    (*Switch to another storage tank with same varnish if storage tank reaches error level.*)
    IF iL_StoragetankAssignmentIndex[iL_Counter] <> 0 THEN
      IF sAdsIkInkStorageTank[iL_StoragetankAssignmentIndex[iL_Counter]].bO_StorageTankError THEN
        FOR iL_Counter2 := 1 TO iCIk_NB_INKSTORAGE_TANK DO
          IF     (iL_StoragetankAssignmentIndex[iL_Counter] <> iL_Counter2)
             AND (  sAdsIkInkStorageTank[iL_StoragetankAssignmentIndex[iL_Counter]].sI_InkParameter.iIndex
                  = sAdsIkInkStorageTank[iL_Counter2].sI_InkParameter.iIndex)
             AND NOT sAdsIkInkStorageTank[iL_Counter2].bO_StorageTankError
          THEN
            sAdsIkHeaderTank[iL_Counter].sI_StoragetankAssignment   .lI_Val := UDINT_TO_DINT(sL_BLK_INKSTORAGE_TANK[iL_Counter2].iBlk_AdsId);
            sAdsIkHeaderTank[iL_Counter].sO_ActStoragetankAssignment.lI_Val := UDINT_TO_DINT(sL_BLK_INKSTORAGE_TANK[iL_Counter2].iBlk_AdsId);
          END_IF
        END_FOR
      END_IF
    END_IF
  
    (*Check assignment of header tank to storage tank*)
    iL_StoragetankAssignmentIndex   [iL_Counter] := 0;
    iL_ActStoragetankAssignmentIndex[iL_Counter] := 0;
  
    FOR iL_Counter2 := 1 TO iCIk_NB_INKSTORAGE_TANK DO
      IF   sAdsIkHeaderTank[iL_Counter].sI_StoragetankAssignment.lI_Val
         = UDINT_TO_DINT(sL_BLK_INKSTORAGE_TANK[iL_Counter2].iBlk_AdsId)
      THEN
        iL_StoragetankAssignmentIndex[iL_Counter] := iL_Counter2;
      END_IF
  
      IF   sAdsIkHeaderTank[iL_Counter].sO_ActStoragetankAssignment.lI_Val
         = UDINT_TO_DINT(sL_BLK_INKSTORAGE_TANK[iL_Counter2].iBlk_AdsId)
      THEN
        iL_ActStoragetankAssignmentIndex[iL_Counter] := iL_Counter2;
      END_IF
    END_FOR

    (*Purge: outflow valve while DeAir*)
    bL_PurgeOutflow2ValveHT[iL_Counter] :=     fb_PurgeController[iCIk_MAP_HEADERTANK_PURGE_CONTR[iL_Counter]].fb_PurgeContr.bI_DeAirSelect[iCIk_MAP_HEADERTANK_PURGE_GROUPIDX[iL_Counter]]
                                           AND fb_PurgeController[iCIk_MAP_HEADERTANK_PURGE_CONTR[iL_Counter]].fb_PurgeContr.bO_Outflow2Valve;

  END_FOR
  
  
  
  FOR iL_Counter := 1 TO iCIk_NB_HEADERTANK DO
    (*Data from assigned storage tank*)
    IF     (iL_ActStoragetankAssignmentIndex[iL_Counter] > 0)
       AND (iL_ActStoragetankAssignmentIndex[iL_Counter] <= iCIk_NB_INKSTORAGE_TANK)
    THEN
      fL_StorageTankLevelLiter := sAdsIkInkStorageTank[iL_ActStoragetankAssignmentIndex[iL_Counter]].fO_StorageTankLevelLiter.fO_Val;
  
      IF sAdsIkInkStorageTank[iL_ActStoragetankAssignmentIndex[iL_Counter]].sI_InkParameter.iTimer = 0 THEN
        IF (sAdsIkInkStorageTank[iL_ActStoragetankAssignmentIndex[iL_Counter]].sI_InkParameter.iColorId >= 254) THEN
          tL_TimeReturnFlow := tL_TimeReturnFlowHt[iL_Counter];
        ELSE
          tL_TimeReturnFlow := UDINT_TO_TIME(lL_TimeReturnFlow * 1000);
        END_IF
      ELSE
        tL_TimeReturnFlow := UDINT_TO_TIME(UINT_TO_UDINT(sAdsIkInkStorageTank[iL_ActStoragetankAssignmentIndex[iL_Counter]].sI_InkParameter.iTimer) * 1000);
        tL_TimeReturnFlowHt[iL_Counter] := tL_TimeReturnFlow;
      END_IF
  
      IF     (iL_StoragetankAssignmentIndex   [iL_Counter] > 0)
         AND (iL_StoragetankAssignmentIndex   [iL_Counter] <= iCIk_NB_INKSTORAGE_TANK)
         AND (iL_ActStoragetankAssignmentIndex[iL_Counter] > 0)
         AND (iL_ActStoragetankAssignmentIndex[iL_Counter] <= iCIk_NB_INKSTORAGE_TANK)
      THEN
        (*Special storage tank with conservation*)
        IF FIND(sAdsIkInkStorageTank[iL_StoragetankAssignmentIndex[iL_Counter]].aO_Name, sC_Config_I.aC_STORAGETANK_CONSERVATION) > 0 THEN
          bL_Compatibility := FALSE;
        ELSE
          iL_ActIndex := sAdsIkInkStorageTank[iL_ActStoragetankAssignmentIndex[iL_Counter]].sI_InkParameter.iIndex + 1;
          
          IF iL_ActIndex > 0 THEN
            bL_Compatibility := sAdsIkInkStorageTank[iL_StoragetankAssignmentIndex[iL_Counter]].sI_InkParameter.bCompatibility[iL_ActIndex];
          ELSE
            bL_Compatibility := FALSE;
          END_IF
        END_IF
      ELSE
        bL_Compatibility := FALSE;
      END_IF
    ELSE
      tL_TimeReturnFlow        := UDINT_TO_TIME(lL_TimeReturnFlow * 1000);
      fL_StorageTankLevelLiter := 0;
      bL_Compatibility         := FALSE;
    END_IF
  
    (*Data from desired storage tank*)
    IF     (iL_StoragetankAssignmentIndex[iL_Counter] > 0)
       AND (iL_StoragetankAssignmentIndex[iL_Counter] <= iCIk_NB_INKSTORAGE_TANK)
    THEN
      IF sAdsIkInkStorageTank[iL_StoragetankAssignmentIndex[iL_Counter]].sI_InkParameter.iTimerFill = 0 THEN
        tL_TimeMaxFill := DINT_TO_TIME(WORD_TO_DINT(sC_Config_I.wC_INKPUMP_MAX_TIME) * 1000);
        wL_TimeMaxFillHt[iL_Counter] := sC_Config_I.wC_INKPUMP_MAX_TIME;
      ELSE
        tL_TimeMaxFill := UDINT_TO_TIME(UINT_TO_UDINT(sAdsIkInkStorageTank[iL_StoragetankAssignmentIndex[iL_Counter]].sI_InkParameter.iTimerFill) * 1000);
        wL_TimeMaxFillHt[iL_Counter] := UINT_TO_WORD(sAdsIkInkStorageTank[iL_StoragetankAssignmentIndex[iL_Counter]].sI_InkParameter.iTimerFill);
      END_IF
    ELSE
      tL_TimeMaxFill := DINT_TO_TIME(WORD_TO_DINT(sC_Config_I.wC_INKPUMP_MAX_TIME) * 1000);
      wL_TimeMaxFillHt[iL_Counter] := sC_Config_I.wC_INKPUMP_MAX_TIME;
    END_IF
  
    tL_TimeBlowOut      := UDINT_TO_TIME(lL_TimeBlowOut      * 1000);
    tL_TimeEmptyCleaner := UDINT_TO_TIME(lL_TimeEmptyCleaner * 1000);
    tL_TimeRefuseFlow   := UDINT_TO_TIME(lL_TimeRefuseFlow   * 1000);

    (*---input---*)
    bL_PurgeDeAirValveRequest[iL_Counter] :=     fb_PurgeController[iCIk_MAP_HEADERTANK_PURGE_CONTR[iL_Counter]].fb_PurgeContr.bI_DeAirSelect[iCIk_MAP_HEADERTANK_PURGE_GROUPIDX[iL_Counter]]
                                             AND fb_PurgeController[iCIk_MAP_HEADERTANK_PURGE_CONTR[iL_Counter]].fb_PurgeContr.bO_DeAirValve;

    fb_Headertank[iL_Counter].pI_sAdsHeadertank            := ADR(sAdsIkHeaderTank[iL_Counter]);
    fb_Headertank[iL_Counter].pI_StorTankAssignIndex       := ADR(iL_StoragetankAssignmentIndex[iL_Counter]);
    fb_Headertank[iL_Counter].pI_ActStorTankAssignIndex    := ADR(iL_ActStoragetankAssignmentIndex[iL_Counter]);
    fb_Headertank[iL_Counter].bI_PurgeActive               := bL_PurgeBusy;
    fb_Headertank[iL_Counter].bI_PurgeValveActive          := fb_PurgeController[iCIk_MAP_HEADERTANK_PURGE_CONTR[iL_Counter]].fbPurgeGroup[iCIk_MAP_HEADERTANK_PURGE_GROUPIDX[iL_Counter]].bO_PurgeReleaseValve;
    fb_Headertank[iL_Counter].bI_DeAirValveRequest         :=    bL_PurgeDeAirValveRequest[iL_Counter]
                                                              OR fb_CirculationInk[iL_Counter].ObHtCloseMencConnectionValve;
    fb_Headertank[iL_Counter].bI_Outflow1ValveRequest      := bL_PurgeOutflow1ValveHT[iL_Counter];
    fb_Headertank[iL_Counter].bI_Outflow2ValveRequest      :=    bL_PurgeOutflow2ValveHT[iL_Counter]
                                                              OR fb_CirculationInk[iL_Counter].ObValveActivation;
    fb_Headertank[iL_Counter].bI_FillPumpConfirmation      := fb_Headertank[iL_Counter].bO_FillPumpRequest;
    fb_Headertank[iL_Counter].bI_CleanerPumpInUse          := bL_CleanerPumpRequest[iCIk_MAP_HEADERTANK_CLEANER_PUMP[iL_Counter]];
    fb_Headertank[iL_Counter].bI_CleanerPumpConfirmation   := bL_CleanerPumpConfirmation[iL_Counter];
    fb_Headertank[iL_Counter].bI_ReturnFlowConfirmation    := bL_ReturnFlowConfirmation[iL_Counter];
    fb_Headertank[iL_Counter].bI_Niveau                    := bIKn_TankInkLevelReached[iL_Counter];
    fb_Headertank[iL_Counter].bI_CleanExec                 := iMachineInk[iCIk_MAP_HEADERTANK_HT_GROUP[iL_Counter]].pCleanExec;
    (*bI_PrintExec is only used to set a message that an exchange with degassed varnish is needed.*)
    fb_Headertank[iL_Counter].bI_PrintExec                 := TRUE;
    fb_Headertank[iL_Counter].tL_TimeWarnExchange          := UDINT_TO_TIME(lL_TimeWarnExchange * 1000 * 60 * 60);  (*[h] => [ms]*)
    fb_Headertank[iL_Counter].fI_StorageTankLevelLiter     := fL_StorageTankLevelLiter;  (*not used yet*)
    fb_Headertank[iL_Counter].bI_Compatibility             := bL_Compatibility;
    fb_Headertank[iL_Counter].StateChange                  := eL_LowestActiveStateChange  [iCIk_MAP_HEADERTANK_HT_GROUP[iL_Counter]];
    fb_Headertank[iL_Counter].StateEmpty                   := eL_LowestActiveStateEmpty   [iCIk_MAP_HEADERTANK_HT_GROUP[iL_Counter]];
    fb_Headertank[iL_Counter].StateFill                    := eL_LowestActiveStateFill    [iCIk_MAP_HEADERTANK_HT_GROUP[iL_Counter]];
    fb_Headertank[iL_Counter].StateFlush                   := eL_LowestActiveStateFlush   [iCIk_MAP_HEADERTANK_HT_GROUP[iL_Counter]];
    fb_Headertank[iL_Counter].StateCleaning                := eL_LowestActiveStateCleaning[iCIk_MAP_HEADERTANK_HT_GROUP[iL_Counter]];

    (*Until now the pump command comes from FB_INK_SUPPLY_UNIT*)
    fb_Headertank[iL_Counter].bI_FillPumpExtern := fb_FillInkVarnish[iL_Counter].bO_EnablePump;

    (*---call---*)
    IF (iL_StoragetankAssignmentIndex[iL_Counter] > 0) THEN
      bL_HeadertankCanEx :=     iMachineInk[iCIk_MAP_HEADERTANK_HT_GROUP[iL_Counter]].pInCappingPos
                            AND iMachineInk[iCIk_MAP_HEADERTANK_HT_GROUP[iL_Counter]].pSeparatorNiveauOk;

      IF FIND(sAdsIkInkStorageTank[iL_StoragetankAssignmentIndex[iL_Counter]].aO_Name, sC_Config_I.aC_STORAGETANK_CONSERVATION) = 0 THEN
        bL_HeadertankFillCanEx := TRUE;
      ELSE
        bL_HeadertankFillCanEx := FALSE;
      END_IF
    ELSE
      bL_HeadertankCanEx     := FALSE;
      bL_HeadertankFillCanEx := FALSE;
    END_IF

    fb_Headertank[iL_Counter].Change  ( bI_CommandCanEx            :=     bL_HeadertankCanEx 
                                                                      AND bCIk_HEADERTANK_CHANGE[iL_Counter]
                                                                      AND NOT bL_FlushingActiveHt[iL_Counter]
                                                                      AND NOT bO_TankCleanerLevelEmpty
                                                                      AND NOT bO_TankRefuseLevelFull
                                                                      AND NOT bL_ChangeActiveOtherHT[iL_Counter]
                                      , tI_TimeRefuse              := tL_TimeRefuseFlow);
    fb_Headertank[iL_Counter].Empty   ( bI_CommandCanEx            :=     bL_HeadertankCanEx
                                                                      AND NOT bL_FlushingActiveHt[iL_Counter]
                                      , bI_ReturnFlowConfirmation  := bL_ReturnFlowConfirmation[iL_Counter]
                                      , tI_TimeReturnFlow          := tL_TimeReturnFlow
                                      , tI_TimeBlowOut             := tL_TimeBlowOut);
    fb_Headertank[iL_Counter].Fill    ( bI_CommandCanEx            :=     bL_HeadertankCanEx 
                                                                      AND bCIk_HEADERTANK_FILL[iL_Counter]
                                                                      (*Storage tank for Conservation must be skiped*)
                                                                      AND bL_HeadertankFillCanEx
                                                                      AND NOT bL_FlushingActiveHt[iL_Counter]
                                                                      // not working if Cleaner is filled: AND (fb_Headertank[iL_Counter].aL_StateCleaner = 'Idle')
                                      , tI_TimeFillMax             := tL_TimeMaxFill);
    fb_Headertank[iL_Counter].Flush   ( bI_CommandCanEx            :=     bL_HeadertankCanEx
                                                                      AND bCIk_HEADERTANK_FLUSH[iL_Counter]
                                                                      AND NOT bL_FlushingActiveHt[iL_Counter]
                                      , tI_TimeFillCleanerMax      := DINT_TO_TIME(WORD_TO_DINT(sC_Config_I.wC_CLEANERPUMP_MAX_TIME) * 1000)
                                      , tI_TimeEmptyCleaner        := tL_TimeEmptyCleaner
                                      , tI_TimeBlowOut             := tL_TimeBlowOut);
    fb_Headertank[iL_Counter].Cleaning( bI_CommandCanEx            :=     bL_HeadertankCanEx 
                                                                      AND NOT bL_FlushingActiveHt[iL_Counter]
                                                                      AND (fb_Headertank[iL_Counter].aL_StateCleaner = 'Idle'));
    fb_Headertank[iL_Counter].Cleaner ( bI_CommandCanEx            :=     bL_HeadertankCanEx 
                                                                      AND (iL_ActStoragetankAssignmentIndex[iL_Counter] = 0)
                                                                      AND (eL_LowestActiveStateEmpty[iCIk_MAP_HEADERTANK_HT_GROUP[iL_Counter]] = eEmptyEnd)
                                                                      AND NOT bL_FlushingActiveHt[iL_Counter]
                                                                      AND NOT sAdsIkHeaderTank[iL_Counter].sI_CommandEmpty.bI_Command
                                                                      AND NOT sAdsIkHeaderTank[iL_Counter].sI_CommandEmpty.bO_CommandExec
                                      , bI_CommandStop             :=    bIDp_StopFillCleaner[iL_Counter]
                                                                      OR bL_FlushingStop
                                      , tI_TimeFillCleanerMax      := DINT_TO_TIME(WORD_TO_DINT(sC_Config_I.wC_CLEANERPUMP_MAX_TIME) * 1000));
    fb_Headertank[iL_Counter].Output();
    fb_Headertank[iL_Counter].Messaging();

    (*---output---*)
    IF fb_Headertank[iL_Counter].bO_PurgeRequest THEN
      bL_PurgeContrRequestHT[iCIk_MAP_HEADERTANK_PURGE_CONTR[iL_Counter]] :=    bL_PurgeContrRequestHT[iCIk_MAP_HEADERTANK_PURGE_CONTR[iL_Counter]]
                                                                             OR fb_Headertank[iL_Counter].bO_PurgeRequest;
    END_IF
    bL_PurgeGroupRequestHT     [iCIk_MAP_HEADERTANK_PURGE_GROUP[iL_Counter]] := fb_Headertank[iL_Counter].bO_PurgeRequest;
    bL_PurgeGroupRequestDeAirHT[iCIk_MAP_HEADERTANK_PURGE_GROUP[iL_Counter]] := fb_Headertank[iL_Counter].bO_PurgeRequestDeAir;
    (*ToDo: iL_Counter passt so eigentlich nicht zu sAdsIkInkPump*)
    sAdsIkInkPump[iCIk_MAP_HEADERTANK_INK_PUMP[iL_Counter]].cO_StatusInkPump.eO_Activ := fb_Headertank[iL_Counter].bO_FillPumpRequest;
  END_FOR

  (*Interface with Motion System*)
  (*PRG_MACHINE.bI_CleanCommandFromInk   := bL_CleanCommandToMachine;*)
  (*PRG_MACHINE.bI_CleanEnable1FromInk   := bL_CleanEnable1ToMachine;*)
  (*PRG_MACHINE.bI_CleanEnable2FromInk   := bL_CleanEnable2ToMachine;*)
  (*PRG_MACHINE.bI_CappingCommandFromInk := bL_CappingCommandToMachine;*)
  bL_CleanCommandToMachine[1]:= FALSE;
  bL_CleanCommandToMachine[2]:= FALSE;
  bL_CleanEnable1ToMachine   := FALSE;
  bL_CleanEnable2ToMachine   := FALSE;
  bL_CappingCommandToMachine := FALSE;
  FOR iL_Counter := 1 TO iCIk_NB_HEADERTANK DO
    bL_CleanCommandToMachine[iCIk_MAP_HEADERTANK_HT_GROUP[iL_Counter]] := bL_CleanCommandToMachine[iCIk_MAP_HEADERTANK_HT_GROUP[iL_Counter]] OR fb_Headertank[iL_Counter].bO_CleanRequest;
    IF fb_Headertank[iL_Counter].bO_CleanRequest THEN
      IF iCIk_MAP_HEADERTANK_INK[iL_Counter] = 1 THEN
        bL_CleanEnable1ToMachine   := TRUE;    
      END_IF
      IF iCIk_MAP_HEADERTANK_INK[iL_Counter] = 2 THEN
        bL_CleanEnable2ToMachine   := TRUE;    
      END_IF
    END_IF
    bL_CappingCommandToMachine := bL_CappingCommandToMachine OR fb_Headertank[iL_Counter].bO_CappingRequest;
  END_FOR
  iMachineInk[1].pCleanCommand := bL_CleanCommandToMachine[1];
  iMachineInk[2].pCleanCommand := bL_CleanCommandToMachine[2];

  (*Command for printline*)
  FOR iL_Counter := 1 TO iCIk_NB_HEADERTANK_GROUP DO
    bO_CommandPrintlineExec[iL_Counter] := FALSE;
 
   (*Change printline*)
    sL_CommandChangePrintline[iL_Counter].bO_CommandCanEx := FALSE;
    FOR iL_Counter2 := 1 TO iCIk_NB_HEADERTANK DO
      IF sAdsIkHeaderTank[iL_Counter2].sI_CommandChange.bO_CommandCanEx THEN
        sL_CommandChangePrintline[iCIk_MAP_HEADERTANK_HT_GROUP[iL_Counter2]].bO_CommandCanEx := TRUE;
      END_IF
    END_FOR
  
    sL_CommandChangePrintline[iL_Counter].bO_CommandExec := FALSE;
    FOR iL_Counter2 := 1 TO iCIk_NB_HEADERTANK DO
      IF    sAdsIkHeaderTank[iL_Counter2].sI_CommandChange.bO_CommandExec 
         OR sAdsIkHeaderTank[iL_Counter2].sI_CommandEmpty .bO_CommandExec
         (*Info needed for fill conservation*)
         OR sAdsIkHeaderTank[iL_Counter2].sI_ActivateCleaner.bO_CommandExec
         OR sAdsIkHeaderTank[iL_Counter2].sI_ActivateCleaner.bI_Command
      THEN
        sL_CommandChangePrintline[iCIk_MAP_HEADERTANK_HT_GROUP[iL_Counter2]].bO_CommandExec := TRUE;
        bO_CommandPrintlineExec  [iCIk_MAP_HEADERTANK_HT_GROUP[iL_Counter2]]                := TRUE;
      END_IF
    END_FOR
  END_FOR

  (*Check assignment of header tank to storage tank*)
  FOR iL_Counter := 1 TO iCIk_NB_HEADERTANK DO
    sAdsIkHeaderTank[iL_Counter].sI_StoragetankAssignment.lI_Val    := 0;
    sAdsIkHeaderTank[iL_Counter].sO_ActStoragetankAssignment.lI_Val := 0;
    FOR iL_Counter2 := 1 TO iCIk_NB_INKSTORAGE_TANK DO
      IF    (iL_StoragetankAssignmentIndex[iL_Counter] = iL_Counter2)
         OR (iL_StoragetankAssignmentIndex[iL_Counter] = UDINT_TO_DINT(sL_BLK_INKSTORAGE_TANK[iL_Counter2].iBlk_AdsId))
      THEN
        sAdsIkHeaderTank[iL_Counter].sI_StoragetankAssignment.lI_Val
          := UDINT_TO_DINT(sL_BLK_INKSTORAGE_TANK[iL_Counter2].iBlk_AdsId);
      END_IF
      IF    (iL_ActStoragetankAssignmentIndex[iL_Counter] = iL_Counter2)
         OR (iL_ActStoragetankAssignmentIndex[iL_Counter] = UDINT_TO_DINT(sL_BLK_INKSTORAGE_TANK[iL_Counter2].iBlk_AdsId))
      THEN
        sAdsIkHeaderTank[iL_Counter].sO_ActStoragetankAssignment.lI_Val
          := UDINT_TO_DINT(sL_BLK_INKSTORAGE_TANK[iL_Counter2].iBlk_AdsId);
      END_IF
    END_FOR
  END_FOR


  (*Cleaner*)
  (******************)
  (*Pump setpoint*)
  wL_StptSpeedCleanInkPumpPercent := LIMIT( lR_MinSpeedFillInkPumpCleaner
                                          , lR_StptSpeedCleanInkPumpCleanerPercent
                                          , lR_MaxSpeedFillInkPumpCleaner);	(*Limitation of setpoint*)
  
  IF (wIDp_AnalogMaxPercentCleaner - wIDp_AnalogMinPercentCleaner) <> 0 THEN
    fL_MFunction := 1.0 * DINT_TO_REAL(lR_AnalogMaxDigitCleaner - lR_AnalogMinDigitCleaner)
                        / DINT_TO_REAL(wIDp_AnalogMaxPercentCleaner - wIDp_AnalogMinPercentCleaner); (*calculation ramp for analog-output of pump*)
  END_IF;
  wL_StptSpeedCleanInkPumpDigit := FC_REAL_TO_WORD(fL_MFunction * wL_StptSpeedCleanInkPumpPercent + DINT_TO_REAL(lR_AnalogMinDigitCleaner));  (*calculated pump speed in digits*)
  
  FOR iL_Counter := 1 TO iCIk_NB_CLEANER_PUMPS DO
    (*---input---*)
    fb_Cleaner[iL_Counter].sI_SystemCmd    := sL_SystemCmd;
    fb_Cleaner[iL_Counter].bI_Acknowledge  := FALSE;  (*not used*)
    fb_Cleaner[iL_Counter].wI_MaxPumpTime  := 0;      (*not used*)
    fb_Cleaner[iL_Counter].wI_SetPointPump := wL_StptSpeedCleanInkPumpDigit;
  
    (*init*)
    bL_CleanerPumpRequest[iL_Counter] := FALSE;
    FOR iL_Counter2 := 1 TO iCIk_NB_HEADERTANK DO
      IF (iCIk_MAP_HEADERTANK_CLEANER_PUMP[iL_Counter2] = iL_Counter) THEN 
        bL_CleanerPumpConfirmation[iL_Counter2] := FALSE;
      END_IF
    END_FOR
  
    FOR iL_Counter2 := 1 TO iCIk_NB_HEADERTANK DO
      IF     (iCIk_MAP_HEADERTANK_CLEANER_PUMP[iL_Counter2] = iL_Counter) 
         AND NOT bL_CleanerPumpRequest[iL_Counter]
      THEN
        bL_CleanerPumpRequest     [iL_Counter]  := fb_Headertank[iL_Counter2].bO_CleanerPumpRequest;
        bL_CleanerPumpConfirmation[iL_Counter2] := fb_Headertank[iL_Counter2].bO_CleanerPumpRequest;
        fb_Cleaner[iL_Counter].bI_PumpRequest   := fb_Headertank[iL_Counter2].bO_CleanerPumpRequest;
      END_IF
    END_FOR
  
    (*---call---*)
    fb_Cleaner[iL_Counter].PumpOption(bI_PumpSetPoint := iCIk_CLEANER_PUMP_SETPOINT[iL_Counter]);
    fb_Cleaner[iL_Counter].Pump();
  END_FOR
  
  
  (*Return flow*)
  (******************)
  FOR iL_Counter := 1 TO iCIk_NB_RETURN_FLOW_UNITS DO
    (*---input---*)
    fb_ReturnFlow[iL_Counter].sI_SystemCmd   := sL_SystemCmd;
    fb_ReturnFlow[iL_Counter].bI_Acknowledge := FALSE;  (*not used*)
    fb_ReturnFlow[iL_Counter].wI_MaxPumpTime := 0;      (*not used*)
  
    (*init*)
    bL_ReturnFlowRequest[iL_Counter]           := FALSE;
    fb_ReturnFlow[iL_Counter].bI_PumpRequest   := FALSE;
    fb_ReturnFlow[iL_Counter].bI_BypassValve   := FALSE;
    (*Reset valves with a delay because pump request is made with a PWM.*)
    IF fb_TonReturnFlowValveDelay[iL_Counter].Q THEN
      fb_ReturnFlow[iL_Counter].bI_RefuseRequest := FALSE;
      FOR iL_Counter2 := 1 TO iCIk_NB_INKSTORAGE_TANK_MAX DO
        fb_ReturnFlow[iL_Counter].bI_StoragetankAssignment[iL_Counter2] := FALSE;
      END_FOR
		END_IF
    FOR iL_Counter2 := 1 TO iCIk_NB_HEADERTANK DO
      IF (iCIk_MAP_HEADERTANK_RETURN_FLOW[iL_Counter2] = iL_Counter) THEN
        bL_ReturnFlowConfirmation[iL_Counter2] := FALSE;
      END_IF
    END_FOR
  
    iL_NbReturnFlowAssignHT[iL_Counter] := 0;
    iL_NbReturnFlowRequest [iL_Counter] := 0;
    bL_ReturnFlowRefuse    [iL_Counter] := FALSE;
    FOR iL_Counter2 := 1 TO iCIk_NB_HEADERTANK DO
      IF     (iCIk_MAP_HEADERTANK_RETURN_FLOW[iL_Counter2] = iL_Counter) 
         (*not needed here because each tank group has it's own return pump
         AND NOT bL_ReturnFlowRequest[iL_Counter] *)
      THEN
        iL_NbReturnFlowAssignHT[iL_Counter] := iL_NbReturnFlowAssignHT[iL_Counter] + 1;
        (*Check number of requests for PWM control of pump*)
        IF    fb_Headertank[iL_Counter2].bO_ReturnFlowPumpRequest 
           OR bL_PurgeDeAirValveRequest[iL_Counter2]
           OR fb_CirculationInk[iL_Counter2].ObPumpActivation
           // is done with a special pump OR bL_FlushingReturnFlowRequest[iL_Counter2]
        THEN
          bL_ReturnFlowRequest     [iL_Counter]      := TRUE;
          bL_ReturnFlowConfirmation[iL_Counter2]     := TRUE;
          bL_ReturnFlowRefuse      [iL_Counter]      :=  bL_ReturnFlowRefuse[iL_Counter] OR fb_Headertank[iL_Counter2].bO_ReturnFlowRefuse;
  
          iL_NbReturnFlowRequest[iL_Counter] := iL_NbReturnFlowRequest[iL_Counter] + 1;
  
          IF     (iL_ActStoragetankAssignmentIndex[iL_Counter2] > 0) 
             AND (iL_ActStoragetankAssignmentIndex[iL_Counter2] <= iCIk_NB_INKSTORAGE_TANK)
          THEN
            fb_ReturnFlow[iL_Counter].bI_StoragetankAssignment[iL_ActStoragetankAssignmentIndex[iL_Counter2]] := TRUE;
          END_IF
        END_IF
      END_IF
    END_FOR

    fb_TonReturnFlowValveDelay[iL_Counter](IN := NOT bL_ReturnFlowRequest[iL_Counter], PT := T#200MS);

    (*PWM control depending on number of requesting HT*)
    IF iL_NbReturnFlowAssignHT[iL_Counter] <> 0 THEN
      fb_TimerReturnFlow[iL_Counter]( bI_Enable    := TRUE
                                    , tI_Frequency := T#25MS
                                    , iI_DutyCycle := (100 * iL_NbReturnFlowRequest[iL_Counter]) / iL_NbReturnFlowAssignHT[iL_Counter]);
    END_IF
    
    IF bL_ReturnFlowRequest[iL_Counter] THEN
      fb_ReturnFlow[iL_Counter].bI_PumpRequest   := bL_ReturnFlowRequest[iL_Counter] AND fb_TimerReturnFlow[iL_Counter].bO_State;
      fb_ReturnFlow[iL_Counter].bI_BypassValve   := FALSE;
      fb_ReturnFlow[iL_Counter].bI_RefuseRequest := bL_ReturnFlowRefuse[iL_Counter];
    END_IF
  
    (*---call---*)
    fb_ReturnFlow[iL_Counter].PumpOption(bI_PumpSetPoint := iCIk_RETURN_FLOW_PUMP_SETPOINT);
    fb_ReturnFlow[iL_Counter].Pump();
    fb_ReturnFlow[iL_Counter].Valves();
    
    (*Return flow valve has negativ logic than output of fb_ReturnFlow*)
    fb_ReturnFlowStorTank[iL_Counter]();
    IF fb_ReturnFlow[iL_Counter].fb_ReturnFlowPump.bOKp_EnablePump THEN
      IF fb_ReturnFlow[iL_Counter].bOKp_ReturnFlowSelRefuse THEN 
        fb_ReturnFlowStorTank[iL_Counter].mDisable(); 
      ELSE 
        fb_ReturnFlowStorTank[iL_Counter].mEnable(); 
      END_IF
    ELSE
      fb_ReturnFlowStorTank[iL_Counter].mDisable(); 
		END_IF
  END_FOR


	(*Fill Ink Varnish*)
	(******************)
  bIDp_EnableMainDgasValve := FALSE;
  FOR iL_Counter := 1 TO iCIk_NB_HEADERTANK DO
    (*---collect conditions---*)
    sL_PumpConditions.bI_SubMencEnabled             := sAdsIkMenc[iCIk_MAP_HEADERTANK_MENC_STA[iL_Counter]].bI_Enable;
    sL_PumpConditions.bI_SubMencOk                  := TRUE;
    sL_PumpConditions.bI_DgasPressOk                := fb_DgasMencContr[iCIk_MAP_HEADERTANK_DGAS[iL_Counter]].pErrorCode = 0;

    sL_PumpConditions.bI_BalancePumpStateOk         := TRUE;
    sL_PumpConditions.bI_BalanceMaintenanceNoExec   := TRUE;
    sL_PumpConditions.bI_WasteBinNotFull            := TRUE;
    sL_PumpConditions.bI_WcStateOk                  := NOT (   bI_InkLevel1WcState
                                                            OR bI_SubPressureWcState[1]
                                                            OR bI_Pressure1WcState);
    sL_PumpConditions.bI_StorTankSetZeroNoExec      := TRUE;
    sL_PumpConditions.bL_HeadertankFillAllowed      := NOT fb_Headertank[iL_Counter].bL_DisableHeadertankFill;

    (*---input---*)
		fb_FillInkVarnish[iL_Counter].sI_SystemCmd         := sL_SystemCmd;
		fb_FillInkVarnish[iL_Counter].sI_InkPumpConditions := sL_PumpConditions;
		fb_FillInkVarnish[iL_Counter].wI_AnalogMaxDigit    := wIDP_AnalogMaxDigitVarnish;
		fb_FillInkVarnish[iL_Counter].wI_AnalogMinDigit    := wIDP_AnalogMinDigitVarnish;
		fb_FillInkVarnish[iL_Counter].bI_EnableAuto        := sAdsIkHeaderTank[iL_Counter].bI_FillModeAuto;
		fb_FillInkVarnish[iL_Counter].bI_EnablePump        :=     (   sAdsIkHeaderTank[iL_Counter].bI_EnableFillInk
                                                               OR fb_Headertank[iL_Counter].bO_FillRequest);
                                                          (*not used, different bahavior     
                                                          AND (   bOKp_EnableStorageTankValve[1]
                                                               OR bOKp_EnableStorageTankValve[2])*)
		fb_FillInkVarnish[iL_Counter].bI_Niveau            := bIKn_TankInkLevelReached[iL_Counter];
		fb_FillInkVarnish[iL_Counter].bI_PumpManu          := sAdsIkHeaderTank[iL_Counter].bI_FillManual;
		fb_FillInkVarnish[iL_Counter].tI_PumpTime          := WORD_TO_TIME(wIDp_PumpTimeOffDelayVarnish);
    fb_FillInkVarnish[iL_Counter].wI_MaxPumpTime       := wL_TimeMaxFillHt[iL_Counter];
    fb_FillInkVarnish[iL_Counter].wI_LevelDelayTime    := sC_Config_I.wC_INKPUMP_LEVELDELAY_TIME;

    IF sAdsIkHeaderTank[iL_Counter].bI_EnableRamp THEN
      fb_Ramp[iL_Counter].II_YAnalogMaxDigit   := IIDp_MaxDigitRampe;
      fb_Ramp[iL_Counter].II_YAnalogMinDigit   := IIDp_MinDigitRampe;
      fb_Ramp[iL_Counter].II_YAnalogMaxPercent := IIDp_MaxPercentRampe;
      fb_Ramp[iL_Counter].II_YAnalogMinPercent := IIDp_MinPercentRampe;
      fb_Ramp[iL_Counter].fI_YAnalogMaxVolt    := fIDp_MaxVoltRampe;
      fb_Ramp[iL_Counter].fI_YAnalogMinVolt    := fIDp_MinVoltRampe;
      fb_Ramp[iL_Counter].II_XTimeRamp         := IIDp_TimeRampe;
  
      fb_Ramp[iL_Counter].bI_EnableRamp        := sAdsIkHeaderTank[iL_Counter].bI_EnableRamp AND sAdsIkHeaderTank[iL_Counter].bI_FillModeAuto;
      fb_Ramp[iL_Counter].bI_StartRamp         := fb_FillInkVarnish[iL_Counter].bO_EnablePump; (*NOT bL_TankInkLevelReachedVarnish[iL_Counter];*)
      (*ToDo: iL_Counter passt so eigentlich nicht zu sAdsIkInkPump*)
      fb_Ramp[iL_Counter].II_SpeedActPercent   := sAdsIkInkPump[iCIk_MAP_HEADERTANK_INK_PUMP[iL_Counter]].sI_InkPumpSpeedSet.lI_Val;
  
      fb_Ramp[iL_Counter]();
  
      fb_FillInkVarnish[iL_Counter].wI_StptInkPumpPercent := DINT_TO_WORD(fb_Ramp[iL_Counter].IO_YPercent);
    ELSE
      (*ToDo: iL_Counter passt so eigentlich nicht zu sAdsIkInkPump*)
      fb_FillInkVarnish[iL_Counter].wI_StptInkPumpPercent := DINT_TO_WORD(sAdsIkInkPump[iCIk_MAP_HEADERTANK_INK_PUMP[iL_Counter]].sI_InkPumpSpeedSet.lI_Val);
    END_IF

		fb_FillInkVarnish[iL_Counter].wI_StptInkPumpPercentMin	:= wIDp_MinSpeedFillInkPumpVarnish;
		fb_FillInkVarnish[iL_Counter].wI_StptInkPumpPercentMax	:= wIDp_MaxSpeedFillInkPumpVarnish;
		fb_FillInkVarnish[iL_Counter]();

    IF fb_FillInkVarnish[iL_Counter].bI_EnablePump AND NOT sAdsIkHeaderTank[iL_Counter].bI_EnableRamp THEN
      wOKp_StptSpeedFillInkPumpVarnish[iL_Counter]	:= fb_FillInkVarnish[iL_Counter].wO_PumpSpeed;
    ELSE
      wOKp_StptSpeedFillInkPumpVarnish[iL_Counter]	:= DINT_TO_WORD(fb_Ramp[iL_Counter].IO_YDigit);
    END_IF
  
    bOKp_EnableFillInkPumpVarnish[iL_Counter] := fb_FillInkVarnish[iL_Counter].bO_EnablePump;

  //bIDp_EnableMainDgasValve := bIDp_EnableMainDgasValve OR sAdsIkHeaderTank[iL_Counter].bI_EnableFillInk;
    bIDp_EnableMainDgasValve := bIDp_EnableMainDgasValve OR fb_Headertank[iL_Counter].bO_FillPumpRequest;

    (*Set CanEx if error*)
    IF fb_FillInkVarnish[iL_Counter].bO_ErrorPumpTime THEN
      sAdsIkHeaderTank[iL_Counter].sI_AckFillInk.bO_CommandCanEx := TRUE;
		ELSE
      sAdsIkHeaderTank[iL_Counter].sI_AckFillInk.bO_CommandCanEx := FALSE;
		END_IF;

		(*Acknowledge fill ink error*)
		IF FC_COMMAND(ADR(sAdsIkHeaderTank[iL_Counter].sI_AckFillInk)) THEN
			fb_FillInkVarnish[iL_Counter].bI_AckFault                  := TRUE;		(*clear fill ink error*)
			sAdsIkHeaderTank[iL_Counter].sI_AckFillInk.bO_CommandCanEx := FALSE;
		ELSE
			fb_FillInkVarnish[iL_Counter].bI_AckFault                  := FALSE;	(*clear fill ink error*)
		END_IF

		(*update ADS status*)
		sAdsIkHeaderTank[iL_Counter].cO_StatusFillInk.eO_Activ       := fb_FillInkVarnish[iL_Counter].bO_FillActiv;
		sAdsIkHeaderTank[iL_Counter].cO_StatusFillInk.eO_SpareBit5   := NOT bIKn_TankInkLevelReached[iL_Counter];
		sAdsIkHeaderTank[iL_Counter].cO_StatusFillInk.eO_SpareBit6   := fb_FillInkVarnish[iL_Counter].bO_EnableValve;
    sAdsIkHeaderTank[iL_Counter].cO_StatusFillInk.eO_SpareBit7   := fb_Ramp[iL_Counter].bO_MaxSpeedReached;

    sAdsIkHeaderTank[iL_Counter].bO_EnableFillInkCanEn           := bCIk_HEADERTANK_EXIST[iL_Counter] AND NOT bL_FlushingActiveHt[iL_Counter];

    (*Messaging in fb_FillInkVarnish only dummy, messaging is now handled by fb_Headertank*)
    fb_Headertank[iL_Counter].bI_Msg[1]  := fb_FillInkVarnish[iL_Counter].fb_Msg[1].bI_Status;
    fb_Headertank[iL_Counter].bI_Msg[2]  := fb_FillInkVarnish[iL_Counter].fb_Msg[2].bI_Status;
    fb_Headertank[iL_Counter].bI_Msg[3]  := fb_FillInkVarnish[iL_Counter].fb_Msg[3].bI_Status;
    fb_Headertank[iL_Counter].bI_Msg[4]  := fb_FillInkVarnish[iL_Counter].fb_Msg[4].bI_Status;
    fb_Headertank[iL_Counter].bI_Msg[5]  := fb_FillInkVarnish[iL_Counter].fb_Msg[5].bI_Status;
    fb_Headertank[iL_Counter].bI_Msg[6]  := fb_FillInkVarnish[iL_Counter].fb_Msg[6].bI_Status;
    fb_Headertank[iL_Counter].bI_Msg[10] := FALSE;
  END_FOR


  (*Circulation ink controller*)
  FOR iL_Counter := 1 TO iCIk_NB_HEADERTANK DO
    fb_CirculationInk[iL_Counter]( IbAxisMovement := PRG_MACHINE.fbMachineComm.bMachineMoving
                                 , IbHeadertankOk :=     sAdsIkHeaderTank[iL_Counter].bI_EnableFillInk                        (*Fill ink is enabled*)
                                                     AND NOT sAdsIkHeaderTank[iL_Counter].sI_CommandChange.bO_CommandExec     (*Execution not active*)
                                                     AND NOT sAdsIkHeaderTank[iL_Counter].sI_CommandEmpty.bO_CommandExec      (*Execution not active*)
                                                     AND NOT sAdsIkHeaderTank[iL_Counter].sI_CommandFlush.bO_CommandExec      (*Execution not active*)
                                                     AND (fb_Headertank[iL_Counter].aL_StateCleaner = 'Idle')                 (*No cleaner filled*)
                                                     AND NOT fb_FillInkVarnish[iL_Counter].bO_ErrorPumpTime                   (*No fill ink error*)
                                                     AND NOT fb_FillInkVarnish[iL_Counter].bO_ErrorLevel                      (*No fill ink error*)
                                                     AND NOT fb_FillInkVarnish[iL_Counter].bO_ErrorPumpMonitoring             (*No fill ink error*)
                                                     AND fb_TempControllerHys[iCIk_MAP_HEADERTANK_TEMP_CONTR[iL_Counter]].pErrorCode = 0
                                 , IbPHTempOk     := NOT PRG_PRINT.stPcFlags[iCIk_MAP_HEADERTANK_INK[iL_Counter]].bTempOutOfRange
                                 );
    bO_HTInkConnectionClose[iL_Counter] := NOT fb_CirculationInk[iL_Counter].ObHtCloseInkConnectionValve;
  END_FOR


  (*Storagetank*)
  (******************)
  FOR iL_Counter := 1 TO iCIk_NB_INKSTORAGE_TANK DO
    (*---input---*)
    fb_Storagetank[iL_Counter].bI_Msg[ 1] := fB_BalanceMsg[iL_Counter,  1].bI_Status;
    fb_Storagetank[iL_Counter].bI_Msg[ 2] := fB_BalanceMsg[iL_Counter,  2].bI_Status;
    fb_Storagetank[iL_Counter].bI_Msg[ 3] := fB_BalanceMsg[iL_Counter,  3].bI_Status;
    fb_Storagetank[iL_Counter].bI_Msg[ 4] := fB_BalanceMsg[iL_Counter,  4].bI_Status;
    fb_Storagetank[iL_Counter].bI_Msg[ 5] := fB_BalanceMsg[iL_Counter,  5].bI_Status;
    fb_Storagetank[iL_Counter].bI_Msg[ 6] := fB_BalanceMsg[iL_Counter,  6].bI_Status;
    fb_Storagetank[iL_Counter].bI_Msg[ 7] := fB_BalanceMsg[iL_Counter,  7].bI_Status;
    fb_Storagetank[iL_Counter].bI_Msg[ 8] := fB_BalanceMsg[iL_Counter,  8].bI_Status;
    fb_Storagetank[iL_Counter].bI_Msg[ 9] := fB_BalanceMsg[iL_Counter,  9].bI_Status;
    fb_Storagetank[iL_Counter].bI_Msg[10] := fB_BalanceMsg[iL_Counter, 10].bI_Status;
    fb_Storagetank[iL_Counter].bI_Msg[11] := fB_BalanceMsg[iL_Counter, 11].bI_Status;
    fb_Storagetank[iL_Counter].bI_Msg[12] := fB_BalanceMsg[iL_Counter, 12].bI_Status;
    fb_Storagetank[iL_Counter].bI_Msg[13] := fB_BalanceMsg[iL_Counter, 13].bI_Status;
    fb_Storagetank[iL_Counter].bI_Msg[14] := fB_BalanceMsg[iL_Counter, 14].bI_Status;
    fb_Storagetank[iL_Counter].bI_Msg[15] := fB_BalanceMsg[iL_Counter, 15].bI_Status;
  
    fb_Storagetank[iL_Counter].sI_SystemCmd       := sL_SystemCmd;
    fb_Storagetank[iL_Counter].pI_sAdsStoragetank := ADR(sAdsIkInkStorageTank[iL_Counter]);
    fb_Storagetank[iL_Counter].bI_Acknowledge     := FALSE;  (*not used*)
    fb_Storagetank[iL_Counter].wI_MaxPumpTime     := 0;      (*not used*)
  
    FOR iL_Counter2 := 1 TO iCIk_NB_INKSTORAGE_TANK_PUMP DO
      fb_Storagetank[iL_Counter].bI_PumpRequest[iL_Counter2] := FALSE;
    END_FOR
  
    bL_HtAssignedToStorage[iL_Counter] := FALSE;
    FOR iL_Counter2 := 1 TO iCIk_NB_HEADERTANK DO
      IF    (iL_ActStoragetankAssignmentIndex[iL_Counter2] = iL_Counter)
         OR (    (iL_StoragetankAssignmentIndex[iL_Counter2] = iL_Counter))
             AND (   sAdsIkHeaderTank[iL_Counter2].sI_CommandChange.bO_CommandExec
                  OR sAdsIkHeaderTank[iL_Counter2].sI_CommandEmpty.bO_CommandExec 
                  OR sAdsIkHeaderTank[iL_Counter2].sI_CommandFill.bO_CommandExec) 
      THEN   
        bL_HtAssignedToStorage[iL_Counter] := TRUE;
      END_IF
  
      IF iL_StoragetankAssignmentIndex[iL_Counter2] = iL_Counter THEN   
        fb_Storagetank[iL_Counter].bI_PumpRequest[iCIk_MAP_HEADERTANK_STORAGE_PUMP[iL_Counter2]]
          := fb_Headertank[iL_Counter2].bO_FillPumpRequest;
        bL_FillPumpConfirmation[iL_Counter2] := fb_Headertank[iL_Counter2].bO_FillPumpRequest;
  
        (*---output---*)
        bIDp_EnableMainDgasValve := bIDp_EnableMainDgasValve OR fb_Headertank[iL_Counter2].bO_FillPumpRequest;
      END_IF
    END_FOR
    fb_Storagetank[iL_Counter].bI_HtAssignedToStorage     := bL_HtAssignedToStorage[iL_Counter];
  
    (*---call---*)
    fb_Storagetank[iL_Counter].PumpOption(bI_PumpSetPoint := iCIk_STORAGE_TANK_PUMP_SETPOINT);
    fb_Storagetank[iL_Counter].Pump();
    fb_Storagetank[iL_Counter].Messaging();
  END_FOR
  
  (*Barcode scanner*)
  (*****************)
  (*---input---*)
  fb_BarcodeStoragetank.bI_Enable := bI_EnableBarcodeScanner;		(*activate communication*)
  FOR iL_Counter := 1 TO iCIk_NB_INKSTORAGE_TANK DO
    fb_BarcodeStoragetank.bI_WeightOk         [iL_Counter] := NOT sAdsIkInkStorageTank[iL_Counter].cO_StatusBalance.eO_Err;
    fb_BarcodeStoragetank.bI_MaintenanceActive[iL_Counter] := sAdsIkInkStorageTank[iL_Counter].sI_EnableMaintenance.bO_CommandExec;
    fb_BarcodeStoragetank.lI_ScannerId        [iL_Counter] := sAdsIkInkStorageTank[iL_Counter].sI_InkParameter.iScannerId;		(*Scanner ID*)
  END_FOR
  
  
  (*Process barcode communication signals*)
  fb_BarcodeStoragetank.bI_AckInit      := bI_Barcode_AckInit;
  fb_BarcodeStoragetank.bI_DataReceived := bI_Barcode_DataRec;
  fb_BarcodeStoragetank.iI_RecvLength   := iI_Barcode_RecDataLength;
  fb_BarcodeStoragetank.cI_RxBuffer     := cI_Barcode_RxBuff;
  fb_BarcodeStoragetank.bI_BufferFull   := bI_Barcode_BufferFull;
  fb_BarcodeStoragetank.bI_FramingFault := bI_Barcode_FramingError;
  fb_BarcodeStoragetank.bI_OverRunError := bI_Barcode_OverRunError;
  
  (*---call---*)
  fb_BarcodeStoragetank();
  
  (*---output---*)
  bO_Barcode_ReqInit                    := fb_BarcodeStoragetank.bO_ReqInit;
  bO_Barcode_AckRec                     := fb_BarcodeStoragetank.bO_DataRetrieved;
  

  (*BALANCE*)
  (***********************************************************************************************)
  IF bCIk_BALANCE_EXISTING THEN
    (*---input---*)
    fb_BalanceLink.bI_Enable := bI_EnableBalanceLink;		(*activate communication*)

    bL_AckFaultGUI := FALSE;
    FOR iL_Counter := 1 TO iCIk_NB_INKBALANCE DO
      fb_BalanceLink.bI_GW_SelectedChannel [iL_Counter] := FC_COMMAND(ADR(sAdsIkInkStorageTank[iL_Counter].sI_EnableBalance));

      fb_BalanceLink.aI_CalibrateFrameText1[iL_Counter] := sAdsIkInkStorageTank[iL_Counter].aI_CalibrateFrameText1;
      fb_BalanceLink.aI_CalibrateFrameText2[iL_Counter] := sAdsIkInkStorageTank[iL_Counter].aI_CalibrateFrameText2;

      bL_AckFaultGUI                                    := bL_AckFaultGUI OR fB_MsgQueueStorage[iL_Counter].bO_ReceiptMessage;
    END_FOR;

	  (*process balance communication link*)
    fb_BalanceLink.fL_CorrectionValue := fI_CorrectionValue;
    fb_BalanceLink.tI_UpdateRate      := INT_TO_TIME(iI_RefreshRate);
    fb_BalanceLink.bI_AckFaultGUI     := bL_AckFaultGUI;

    (*---call---*)
    fb_BalanceLink();

    (*---output---*)
    (*process balance communication signals*)
    fb_BalanceLink.bI_AckInit      := bI_Balance_AckInit;
    bO_Balance_ReqInit             := fb_BalanceLink.bO_ReqInit;

    fb_BalanceLink.bI_AckSend      := bI_Balance_AckSend;
    bO_Balance_ReqSend             := fb_BalanceLink.bO_SendReq;

    fb_BalanceLink.bI_DataReceived := bI_Balance_DataRec;
    bO_Balance_AckRec              := fb_BalanceLink.bO_DataRetrieved;

    fb_BalanceLink.iI_RecvLength   := iI_Balance_RecDataLength;
    iO_Balance_SendDataLength      := fb_BalanceLink.iO_SendLength;

    FOR iL_Counter := 0 TO 49 DO
      fb_BalanceLink.cI_RxBuffer[iL_Counter]  := UINT_TO_BYTE(cI_Balance_RxBuffWord[iL_Counter]);
      cO_Balance_TxBuffWord[iL_Counter]       := BYTE_TO_UINT(fb_BalanceLink.cO_TxBuffer[iL_Counter]);
    END_FOR;

    FOR iL_Counter := 1 TO iCIk_NB_INKBALANCE DO
      fb_Balance[iL_Counter].fI_StorageTank_ActualLvl
        :=   fb_BalanceLink.fO_Readings[iL_Counter]
           * sAdsIkInkStorageTank[iL_Counter].sI_CorrectionValue.fI_Val;
    END_FOR;

    (*process balance controller inputs*)
    FOR iL_Counter :=1 TO iCIk_NB_INKBALANCE DO
      (*---input---*)
      fb_Balance[iL_Counter].bI_Enable                 := sAdsIkInkStorageTank[iL_Counter].sI_EnableBalance.bI_Command;
      fb_Balance[iL_Counter].bI_MaintenanceOP          := sAdsIkInkStorageTank[iL_Counter].sI_EnableMaintenance.bI_Command;
      fb_Balance[iL_Counter].lI_MaintenanceTimeout     := FC_SET_VAR_DINT(ADR(sAdsIkInkStorageTank[iL_Counter].sI_MaintenanceTimeout.lI_Val));
      fb_Balance[iL_Counter].bI_SetZero                := sAdsIkInkStorageTank[iL_Counter].bI_SetZero (*AND sAdsIkInkStorageTank[iL_Counter].bO_SetZeroCanEx*);
      fb_Balance[iL_Counter].fI_StorageTank_WarningLvl := sAdsIkInkStorageTank[iL_Counter].sI_WarningLevelSet.fI_Val;
      fb_Balance[iL_Counter].fI_StorageTank_ErrorLvl   := sAdsIkInkStorageTank[iL_Counter].sI_ErrorlevelSet.fI_Val;
      fb_Balance[iL_Counter].fI_StorageTank_ActualLvl  :=   fb_BalanceLink.fO_Readings[iL_Counter]
                                                          * sAdsIkInkStorageTank[iL_Counter].sI_CorrectionValue.fI_Val;
      fb_Balance[iL_Counter].bI_AckFaultGUI            := fB_MsgQueueStorage[iL_Counter].bO_ReceiptMessage;
      IF sAdsIkInkStorageTank[iL_Counter].sI_InkParameter.sDensity.fI_Val = 0 THEN
        FB_Balance[iL_Counter].fI_Density              := sAdsIkInkStorageTank[iL_Counter].sI_InkDensitySet.fI_Val;
      ELSE
        FB_Balance[iL_Counter].fI_Density              := sAdsIkInkStorageTank[iL_Counter].sI_InkParameter.sDensity.fI_Val;
      END_IF

      (*---call---*)
      fb_Balance[iL_Counter]();

      sAdsIkInkStorageTank[iL_Counter].bO_SetZeroExec	 :=	sAdsIkInkStorageTank[iL_Counter].bI_SetZero;	(*command feedback*)
    END_FOR;

    (*---output---*)
    (*process balance controller outputs*)
    FOR iL_Counter := 1 TO iCIk_NB_INKBALANCE DO
      (*get balance feedback*)
      IF fb_Balance[iL_Counter].bI_Enable THEN
        IF FB_Balance[iL_Counter].fO_MeasuredQuantity > 0 THEN
          sAdsIkInkStorageTank[iL_Counter].fO_StorageTankLevelLiter.fO_Val := FB_Balance[iL_Counter].fO_MeasuredQuantity;
  
          IF sAdsIkInkStorageTank[iL_Counter].fO_StorageTankSize <> 0 THEN
            sAdsIkInkStorageTank[iL_Counter].fO_StorageTankLevelPercent.fO_Val := (  FB_Balance[iL_Counter].fO_MeasuredQuantity
                                                                                   / sAdsIkInkStorageTank[iL_Counter].fO_StorageTankSize) * 100;
          END_IF;
        ELSE  (*Storage tank is removed from balance*)
          sAdsIkInkStorageTank[iL_Counter].fO_StorageTankLevelLiter.fO_Val   := 0;
          sAdsIkInkStorageTank[iL_Counter].fO_StorageTankLevelPercent.fO_Val := 0;
        END_IF;

        sAdsIkInkStorageTank[iL_Counter].sI_EnableMaintenance.bO_CommandExec := fb_Balance[iL_Counter].bO_MaintenanceExec;
        sAdsIkInkStorageTank[iL_Counter].sO_MaintenanceTimeAct.lO_Val        := fb_Balance[iL_Counter].lO_MaintenanceRemTime;

        sAdsIkInkStorageTank[iL_Counter].bO_SetZeroExec                      := fb_Balance[iL_Counter].bO_SetZero;

        (*StorageTank states*)
        sAdsIkInkStorageTank[iL_Counter].cO_StatusStorageTank.eO_Warn        := (fb_Balance[iL_Counter].eO_StorageState = eWarning);
        sAdsIkInkStorageTank[iL_Counter].bO_StorageTankWarning               := (fb_Balance[iL_Counter].eO_StorageState = eWarning);
        sAdsIkInkStorageTank[iL_Counter].cO_StatusStorageTank.eO_Err         := (fb_Balance[iL_Counter].eO_StorageState = eError);
        sAdsIkInkStorageTank[iL_Counter].bO_StorageTankError                 := (fb_Balance[iL_Counter].eO_StorageState = eError);

        (*Balance states*)
        sAdsIkInkStorageTank[iL_Counter].cO_StatusBalance.eO_Warn            := (fb_Balance[iL_Counter].eO_BalanceState = eWarning);
        sAdsIkInkStorageTank[iL_Counter].cO_StatusBalance.eO_Err             := (fb_Balance[iL_Counter].eO_BalanceState = eError);
      END_IF;

      sAdsIkInkStorageTank[iL_Counter].cO_StatusBalance.eO_Enable            := fb_Balance[iL_Counter].bI_Enable;

      sAdsIkInkStorageTank[iL_Counter].sI_EnableMaintenance.bO_CommandCanEx  :=     sAdsIkInkStorageTank[iL_Counter].sI_EnableBalance.bI_Command
                                                                                AND NOT sAdsIkInkStorageTank[iL_Counter].sI_EnableMaintenance.bI_Command
                                                                                AND NOT sAdsIkInkStorageTank[iL_Counter].sI_EnableMaintenance.bO_CommandExec;
(*      bL_MessageWarning[iL_Counter] := (   sAdsIkInkStorageTank[iL_Counter].bO_StorageTankWarning
                                        OR (    sAdsIkInkStorageTank[iL_Counter].bO_StorageTankError
                                            AND NOT sAdsIkInkStorageTank[iL_Counter].bI_EnableStorageTank));*)
      bL_MessageWarning[iL_Counter] := (    sAdsIkInkStorageTank[iL_Counter].bO_StorageTankWarning
                                        AND sAdsIkInkStorageTank[iL_Counter].bI_EnableStorageTank);
      bL_MessageError  [iL_Counter] := (    sAdsIkInkStorageTank[iL_Counter].bO_StorageTankError
                                        AND sAdsIkInkStorageTank[iL_Counter].bI_EnableStorageTank);
    END_FOR; (*FOR iL_Counter := 1 TO iCIk_NB_INKBALANCE DO*)

    FOR iL_Counter := 1 TO iCIk_NB_INKSTORAGE_TANK DO
      (*Storage Messages*)
      fB_BalanceMsgHandler[iL_Counter]();	(*Call to check for blocked access*)

      fb_BalanceMsg[iL_Counter, 1](bI_Status := fb_BalanceLink.wO_ErrorCodeChannel[iL_Counter].1);
      fb_BalanceMsg[iL_Counter, 2](bI_Status := fb_BalanceLink.wO_ErrorCodeChannel[iL_Counter].2);
      fb_BalanceMsg[iL_Counter, 3](bI_Status := fb_BalanceLink.wO_ErrorCodeChannel[iL_Counter].3);
      fb_BalanceMsg[iL_Counter, 4](bI_Status := fb_BalanceLink.wO_ErrorCodeChannel[iL_Counter].4);
      fb_BalanceMsg[iL_Counter, 5](bI_Status := FALSE);
      fb_BalanceMsg[iL_Counter, 6](bI_Status := FALSE);
      fb_BalanceMsg[iL_Counter, 7](bI_Status := FALSE);
      fb_BalanceMsg[iL_Counter, 8](bI_Status := bL_MessageWarning[iL_Counter]);
      fb_BalanceMsg[iL_Counter, 9](bI_Status := bL_MessageError  [iL_Counter]);
      fb_BalanceMsg[iL_Counter,10](bI_Status := FALSE);
      fb_BalanceMsg[iL_Counter,11](bI_Status := FALSE);  (*InkStorageTankMixerNotWorking*)
      (*Storage tank level info message*)
      fb_BalanceMsg[iL_Counter,12](bI_Status :=     (   sAdsIkInkStorageTank[iL_Counter].bO_StorageTankWarning
                                                     OR sAdsIkInkStorageTank[iL_Counter].bO_StorageTankError)
                                                AND NOT sAdsIkInkStorageTank[iL_Counter].cO_StatusStorageTank.eO_Activ);
      fB_BalanceMsg[iL_Counter,13](bI_Status :=     fb_BarcodeStoragetank.bO_LabelScanNeeded[iL_Counter]
                                                AND sAdsIkInkStorageTank[iL_Counter].cO_StatusStorageTank.eO_Activ);
      fB_BalanceMsg[iL_Counter,14](bI_Status :=     fb_BarcodeStoragetank.bO_LabelScanFalse [iL_Counter]
                                                AND sAdsIkInkStorageTank[iL_Counter].cO_StatusStorageTank.eO_Activ);
      fB_BalanceMsg[iL_Counter,15](bI_Status :=     NOT fb_Storagetank[iL_Counter].bI_HtAssignedToStorage
                                                AND sAdsIkInkStorageTank[iL_Counter].cO_StatusStorageTank.eO_Activ);

      fb_MsgQueueStorage[iL_Counter]();

    END_FOR;
  END_IF; (*IF bCIk_BALANCE_EXISTING THEN*)

  (*Set fO_StorageTankLevelPercent of conservation tank with bO_TankCleanerLevelEmpty*)
  IF bO_TankCleanerLevelEmpty THEN
    sAdsIkInkStorageTank[iCIk_NB_INKSTORAGE_TANK].fO_StorageTankLevelPercent.fO_Val := 0;
  ELSE
    sAdsIkInkStorageTank[iCIk_NB_INKSTORAGE_TANK].fO_StorageTankLevelPercent.fO_Val := 100;
END_IF
  
END_IF; (*Else when init Ok*)


(*Global status*)
bO_InkSystemOk :=     bO_VacuumOk
                  AND bO_TemperatureOk
                //AND bO_StorageTankOk
                  AND (NOT bO_CommandPrintlineExec[1] OR NOT bL_Engaged[1])
                  AND (NOT bO_CommandPrintlineExec[2] OR NOT bL_Engaged[2]);

PRG_PRINT.bI_PuStopByInk := (bO_CommandPrintlineExec[1] AND bL_Engaged[1]) OR (bO_CommandPrintlineExec[2] AND bL_Engaged[2]);

IF sL_SystemCmd.bSleep THEN
  bO_InkStorageTankOk := TRUE;
ELSE
  bO_InkStorageTankOk := FALSE;
  FOR iL_Counter := 1 TO iCIk_NB_INKSTORAGE_TANK DO
    IF bCIk_INKSTORAGE_TANK_EXIST[iL_Counter] THEN
      bO_InkStorageTankOk := bO_InkStorageTankOk OR sAdsIkInkStorageTank[iL_Counter].bI_EnableStorageTank;
    END_IF;
  END_FOR;
END_IF;

(*WcState: 0 = Data valid, 1 = Data invalid*)
bO_TotalWcState     :=     bI_Pressure1WcState
                        OR bI_Pressure2WcState
                        OR bI_SubPressureWcState[1]
                        OR bI_Temperature1WcState
                        OR bI_InkLevel1WcState;


(********************************* END OF PRG ****************************************************)

ACTION AutoFlushingDevice:
IF aI_FlushingSafePattern = 'SAFE' THEN
  bL_FlushingUnlock      := TRUE;
ELSE
  aI_FlushingSafePattern := 'LOCKED';
  bL_FlushingUnlock      := FALSE;
END_IF;
fb_FTrigFlushingActive(CLK:= bL_FlushingActive);
fb_TonFlushingUnlock(IN := bL_FlushingUnlock AND (iL_FlushingState = 0), PT := T#180S);
IF fb_TonFlushingUnlock.Q OR fb_FTrigFlushingActive.Q THEN
  aI_FlushingSafePattern := 'LOCKED';
  bL_FlushingHtEmpty     := FALSE;
END_IF

fb_FlushingReturnFlowTimer( bI_Reset    := (iL_FlushingState = 0)
                          , bI_In       :=    fb_ReturnFlow[iCIk_MAP_HEADERTANK_RETURN_FLOW[PRG_INK.iL_SelHeaderTankFlushing]].fb_ReturnFlowPump.bOKp_EnablePump
                                           OR bO_FlushingReturnPump[iCIk_MAP_HEADERTANK_RETURN_FLOW[PRG_INK.iL_SelHeaderTankFlushing]]
                          , lIO_Seconds := lL_OpCounterReturnFlowSeconds
                          , lIO_Cycles  := lL_OpCounterReturnFlowCycles);

(*Return if function is not unlocked.*)
IF NOT bL_FlushingUnlock THEN
  RETURN;
END_IF

CASE iL_FlushingState OF
0:  (*Idle*)
  aL_FlushingState := 'Idle';

  IF     bL_FlushingActivate 
     AND bL_FlushingHtEmpty 
     AND sAdsIkHeaderTank[PRG_INK.iL_SelHeaderTankFlushing].sI_ActivateCleaner.bO_CommandCanEx
     AND NOT sAdsIkHeaderTank[PRG_INK.iL_SelHeaderTankFlushing].bI_EnableFillInk
  THEN
    bL_FlushingActive := TRUE;

    iL_FlushingState  := 1;
  ELSE
    bL_FlushingStop     := FALSE;
    bL_FlushingActivate := FALSE;
    bL_FlushingActive   := FALSE;
    bL_FlushingActiveHt         [PRG_INK.iL_SelHeaderTankFlushing] := FALSE;
    bL_FlushingReturnFlowRequest[PRG_INK.iL_SelHeaderTankFlushing] := FALSE;
    sAdsIkHeaderTank[PRG_INK.iL_SelHeaderTankFlushing].sI_ActivateCleaner.bI_Command := FALSE;
	END_IF

1:  (*Start fill cleaner*)
  aL_FlushingState := 'Start fill cleaner';

  sAdsIkHeaderTank[PRG_INK.iL_SelHeaderTankFlushing].sI_ActivateCleaner.bI_Command := TRUE;
  
  IF sAdsIkHeaderTank[PRG_INK.iL_SelHeaderTankFlushing].sI_ActivateCleaner.bO_CommandExec THEN
    sAdsIkHeaderTank[PRG_INK.iL_SelHeaderTankFlushing].sI_ActivateCleaner.bI_Command := FALSE;
    bL_FlushingActiveHt[PRG_INK.iL_SelHeaderTankFlushing] := TRUE;

    iL_FlushingState := 2;
	END_IF
  
  IF bL_FlushingStop THEN
    sAdsIkHeaderTank[PRG_INK.iL_SelHeaderTankFlushing].sI_ActivateCleaner.bI_Command := FALSE;

    iL_FlushingState := 5;
	END_IF
  
2:  (*Fill cleaner*)
  aL_FlushingState := 'Fill cleaner';

  IF NOT sAdsIkHeaderTank[PRG_INK.iL_SelHeaderTankFlushing].sI_ActivateCleaner.bO_CommandExec THEN
    iL_FlushingState := 3;
	END_IF
  
  IF bL_FlushingStop THEN
    iL_FlushingState := 5;
	END_IF
  
3:  (*Start empty cleaner*)
  aL_FlushingState := 'Start empty cleaner';

  bL_FlushingReturnFlowRequest[PRG_INK.iL_SelHeaderTankFlushing] := TRUE;
  
  IF    fb_ReturnFlow[iCIk_MAP_HEADERTANK_RETURN_FLOW[PRG_INK.iL_SelHeaderTankFlushing]].fb_ReturnFlowPump.bOKp_EnablePump 
     OR bO_FlushingReturnPump[iCIk_MAP_HEADERTANK_RETURN_FLOW[PRG_INK.iL_SelHeaderTankFlushing]]
  THEN
    iL_FlushingState := 4;
	END_IF

  IF bL_FlushingStop THEN
    bL_FlushingReturnFlowRequest[PRG_INK.iL_SelHeaderTankFlushing] := FALSE;

    iL_FlushingState := 5;
	END_IF
  
4:  (*Empty cleaner*)
  aL_FlushingState := 'Empty cleaner';

  IF lL_OpCounterReturnFlowSeconds >= lL_TimeFlushingReturnFlow THEN
    bL_FlushingReturnFlowRequest[PRG_INK.iL_SelHeaderTankFlushing] := FALSE;
    bL_FlushingActiveHt         [PRG_INK.iL_SelHeaderTankFlushing] := FALSE;

    iL_FlushingState := 0;
	END_IF

  IF bL_FlushingStop THEN
    bL_FlushingReturnFlowRequest[PRG_INK.iL_SelHeaderTankFlushing] := FALSE;

    iL_FlushingState := 5;
	END_IF
  
5:  (*Abort*)
  aL_FlushingState := 'Abort';

  IF     NOT sAdsIkHeaderTank[PRG_INK.iL_SelHeaderTankFlushing].sI_ActivateCleaner.bO_CommandExec
     AND (   NOT fb_ReturnFlow[iCIk_MAP_HEADERTANK_RETURN_FLOW[PRG_INK.iL_SelHeaderTankFlushing]].fb_ReturnFlowPump.bOKp_EnablePump
          OR NOT bO_FlushingReturnPump[iCIk_MAP_HEADERTANK_RETURN_FLOW[PRG_INK.iL_SelHeaderTankFlushing]])
  THEN
    bL_FlushingStop     := FALSE;
    bL_FlushingActivate := FALSE;

    iL_FlushingState := 0;
	END_IF

END_CASE
END_ACTION

ACTION Init:
(*************************************************************************************************)
(* --- Module preprarations --- *)


(*GENERAL*)
(*************************************************************************************************)
(*System init*)
CASE cL_State OF

  cL_INIT : 		(*First init*)

                // Get system reference
                ISystemBase := PRG_SYSTEMBASE.getSystemBaseInterface();
                IF ISystemBase = 0 THEN RETURN; END_IF
                // Wait until system(base) is booted
                IF ISystemBase.bBooting THEN RETURN; END_IF
                
                // Command / Status interface
                PRG_SYSTEMBASE.getSystemStatusInterface(iSystemStatus=>iSystemStatus);
                PRG_SYSTEMBASE.getSystemCmdInterface(iSystemCmd=>iSystemCmd);
                
                // Build mapping information for ADS
                Mapping();
                
                // Register module to system
                pModuleDef := ISystemBase.regModule(
                  pAdsInfo:=ADR(sC_Ads_Info),
                  pMapInfo:=ADR(sMappingInfo)
                );
                IF pModuleDef = 0 THEN RETURN; END_IF

                Fb_RegToAry.iI_ActElem := 0;   (*init module's block mapping array*)
                Fb_RegToAry.sI_Parent := FC_CREATE_ARYPTR(ADR(sL_MOD_MAP), SIZEOF(sL_MOD_MAP)/SIZEOF(sL_MOD_MAP[1]), SIZEOF(sL_MOD_MAP[1]));

                iMachineInk[1] := PRG_MACHINE.fb_InterfaceMachineInk[1];
                iMachineInk[2] := PRG_MACHINE.fb_InterfaceMachineInk[2];

                cL_State := cL_INIT_PRG;

  cL_INIT_PRG :	(*Program call init*)

                FOR iL_CounterDgas := 1 TO iCIk_NB_DGAS DO
                  ;
                END_FOR;

                FOR iL_CounterMenc := 1 TO iCIk_NB_MENC DO
                  ;
                END_FOR

                FOR iL_CounterSubMenc := 1 TO iCIk_NB_SUB_MENC DO
                  ;
                END_FOR

                bL_RemVar_Init := TRUE;    (* Write variables by remanent variables *)
                RemVar();

                cL_State := cL_INIT_OK;

  cL_INIT_OK: 	(*First init ok*)
                bO_InitOk := TRUE;

END_CASE;



(*************************************************************************************************)
(*ADS Structures Init*)
(*************************************************************************************************)

(*INK TABLE*)
(*************************************************************************************************)
sL_InkTable[1].iI_ColorID := 0; sL_InkTable[1].aI_ColorName := sC_Config_I.aC_HEADERTANK_NAME_DETAIL[1]; sL_InkTable[1].lI_ColorRGB := 16#FFFFFF;
sL_InkTable[2].iI_ColorID := 0; sL_InkTable[2].aI_ColorName := sC_Config_I.aC_HEADERTANK_NAME_DETAIL[2]; sL_InkTable[2].lI_ColorRGB := 16#FFFFFF;
sL_InkTable[3].iI_ColorID := 1; sL_InkTable[3].aI_ColorName := sC_Config_I.aC_HEADERTANK_NAME_DETAIL[3]; sL_InkTable[3].lI_ColorRGB := 16#FFFFFF;
sL_InkTable[4].iI_ColorID := 1; sL_InkTable[4].aI_ColorName := sC_Config_I.aC_HEADERTANK_NAME_DETAIL[4]; sL_InkTable[4].lI_ColorRGB := 16#FFFFFF;


(*DEGASSING*)
(*************************************************************************************************)
(*Pneumatic Controller Board CB1*)
(*generate block ads name*)
FOR iL_Counter := 1 TO iCIk_NB_DGAS DO
  aL_Name := sC_Config_I.aC_DGAS_NAME;
  IF sC_Config_I.aC_DGAS_NAME_DETAIL[iL_Counter] <> '' THEN
    aL_Name := CONCAT(aL_Name, CONCAT(' - ', sC_Config_I.aC_DGAS_NAME_DETAIL[iL_Counter]));
  ELSE
    aL_Name := CONCAT(aL_Name, INT_TO_STRING(iL_Counter));
  END_IF
  sAdsIkDgas[iL_Counter].aO_Name := aL_Name;
END_FOR;

sAdsIkDgas[eIk_DGAS1].sI_PressSet.aC_Type := sC_Config_I.aC_DGAS1_PRESS_TYPE;
sAdsIkDgas[eIk_DGAS1].sI_PressSet.aC_Unit := sC_Config_I.aC_DGAS1_PRESS_UNIT;
sAdsIkDgas[eIk_DGAS1].sI_PressSet.fC_Min  := sC_Config_I.fL_DGAS1_PRESS_SET_MIN;
sAdsIkDgas[eIk_DGAS1].sI_PressSet.fC_Max  := sC_Config_I.fL_DGAS1_PRESS_SET_MAX;

sAdsIkDgas[eIk_DGAS1].sO_PressAct.aC_Type := sC_Config_I.aC_DGAS1_PRESS_TYPE;
sAdsIkDgas[eIk_DGAS1].sO_PressAct.aC_Unit := sC_Config_I.aC_DGAS1_PRESS_UNIT;
sAdsIkDgas[eIk_DGAS1].sO_PressAct.fC_Min  := sC_Config_I.fL_DGAS1_PRESS_ACT_MIN;
sAdsIkDgas[eIk_DGAS1].sO_PressAct.fC_Max  := sC_Config_I.fL_DGAS1_PRESS_ACT_MAX;

sAdsIkDgas[eIk_DGAS1].sI_AckPression.bO_CommandExist := TRUE;


(*MENISCUS*)
(*************************************************************************************************)
(*generate block ads name*)
FOR iL_Counter := 1 TO iCIk_NB_MENC DO
  aL_Name := sC_Config_I.aC_MENC_NAME;
  IF sC_Config_I.aC_MENC_NAME_DETAIL[iL_Counter] <> '' THEN
    aL_Name := CONCAT(aL_Name, CONCAT(' - ', sC_Config_I.aC_MENC_NAME_DETAIL[iL_Counter]));
  ELSE
    aL_Name := CONCAT(aL_Name, INT_TO_STRING(iL_Counter));
  END_IF
  sAdsIkMenc[iL_Counter].aO_Name := aL_Name;

  sAdsIkMenc[iL_Counter].sI_PressSet.aC_Type := sC_Config_I.aC_MENC_PRESS_TYPE;
  sAdsIkMenc[iL_Counter].sI_PressSet.aC_Unit := sC_Config_I.aC_MENC_PRESS_UNIT;
  sAdsIkMenc[iL_Counter].sI_PressSet.fC_Min  := sC_Config_I.fL_MENC_PRESS_SET_MIN;
  sAdsIkMenc[iL_Counter].sI_PressSet.fC_Max  := sC_Config_I.fL_MENC_PRESS_SET_MAX;

  sAdsIkMenc[iL_Counter].sO_PressAct.aC_Type := sC_Config_I.aC_MENC_PRESS_TYPE;
  sAdsIkMenc[iL_Counter].sO_PressAct.aC_Unit := sC_Config_I.aC_MENC_PRESS_UNIT;
  sAdsIkMenc[iL_Counter].sO_PressAct.fC_Min  := sC_Config_I.fL_MENC_PRESS_ACT_MIN;
  sAdsIkMenc[iL_Counter].sO_PressAct.fC_Max  := sC_Config_I.fL_MENC_PRESS_ACT_MAX;

  sAdsIkMenc[iL_Counter].sI_AckPression.bO_CommandExist := TRUE;
END_FOR;


(*SUB MENISCUS*)
(*************************************************************************************************)
(*Sub meniscus starts behind the meniscus*)
(*generate block ads name*)
FOR iL_CounterSubMenc := 1 TO iCIk_NB_SUB_MENC DO
  aL_Name := sC_Config_I.aC_SUB_MENC_NAME;
  IF sC_Config_I.aC_SUB_MENC_NAME_DETAIL[iL_CounterSubMenc] <> '' THEN
    aL_Name := CONCAT(aL_Name, CONCAT(' - ', sC_Config_I.aC_SUB_MENC_NAME_DETAIL[iL_CounterSubMenc]));
  ELSE
    aL_Name := CONCAT(aL_Name, INT_TO_STRING(iCIk_NB_MENC + iL_CounterSubMenc));
  END_IF
  sAdsIkMenc[iCIk_NB_MENC + iL_CounterSubMenc].aO_Name := aL_Name;

  sAdsIkMenc[iCIk_NB_MENC + iL_CounterSubMenc].sI_PressSet.aC_Type := sC_Config_I.aC_SUB_MENC_PRESS_TYPE;
  sAdsIkMenc[iCIk_NB_MENC + iL_CounterSubMenc].sI_PressSet.aC_Unit := sC_Config_I.aC_SUB_MENC_PRESS_UNIT;
  sAdsIkMenc[iCIk_NB_MENC + iL_CounterSubMenc].sI_PressSet.fC_Min  := sC_Config_I.fL_SUB_MENC_PRESS_SET_MIN;
  sAdsIkMenc[iCIk_NB_MENC + iL_CounterSubMenc].sI_PressSet.fC_Max  := sC_Config_I.fL_SUB_MENC_PRESS_SET_MAX;

  sAdsIkMenc[iCIk_NB_MENC + iL_CounterSubMenc].sO_PressAct.aC_Type := sC_Config_I.aC_SUB_MENC_PRESS_TYPE;
  sAdsIkMenc[iCIk_NB_MENC + iL_CounterSubMenc].sO_PressAct.aC_Unit := sC_Config_I.aC_SUB_MENC_PRESS_UNIT;
  sAdsIkMenc[iCIk_NB_MENC + iL_CounterSubMenc].sO_PressAct.fC_Min  := sC_Config_I.fL_SUB_MENC_PRESS_ACT_MIN;
  sAdsIkMenc[iCIk_NB_MENC + iL_CounterSubMenc].sO_PressAct.fC_Max  := sC_Config_I.fL_SUB_MENC_PRESS_ACT_MAX;

  sAdsIkMenc[iCIk_NB_MENC + iL_CounterSubMenc].sI_AckPression.bO_CommandExist := TRUE;

  //sAdsIkMenc[iCIk_NB_MENC + iL_CounterSubMenc].iO_ColorId          := x;
END_FOR;


(*PURGE*)
(*************************************************************************************************)
(*generate block ads name*)
FOR iL_Counter := 1 TO iCIk_NB_PURGE_CONTR DO
  aL_Name := sC_Config_I.aC_PURGE_NAME;
  IF sC_Config_I.aC_PURGE_NAME_DETAIL[iL_Counter] <> '' THEN
    aL_Name := CONCAT(aL_Name, CONCAT(' - ', sC_Config_I.aC_PURGE_NAME_DETAIL[iL_Counter]));
  ELSE
    aL_Name := CONCAT(aL_Name, INT_TO_STRING(iL_Counter));
  END_IF
  sAdsIkPurgeController[iL_Counter].aO_Name := aL_Name;

  sAdsIkPurgeController[iL_Counter].sI_ActivatePurge.bO_CommandCanEx := TRUE;
  sAdsIkPurgeController[iL_Counter].sI_ActivatePurge.bO_CommandExist := TRUE;
END_FOR;

FOR iL_Counter := 1 TO iCIk_NB_PURGE_GROUP DO
  (*generate block ads name*)
  aL_Name := sC_Config_I.aC_PURGE_GROUP_NAME;
  IF sC_Config_I.aC_PURGE_GROUP_NAME_DETAIL[iL_Counter] <> '' THEN
    aL_Name := CONCAT(aL_Name, CONCAT(' - ', sC_Config_I.aC_PURGE_GROUP_NAME_DETAIL[iL_Counter]));
  ELSE
    aL_Name := CONCAT(aL_Name, INT_TO_STRING(iL_Counter));
  END_IF
  sAdsIkPurgeGroup[iL_Counter].aO_Name := aL_Name;

  sAdsIkPurgeGroup[iL_Counter].cO_Status.eO_Avbl      := TRUE;
  sAdsIkPurgeGroup[iL_Counter].cO_ValveStatus.eO_Avbl := TRUE;
END_FOR


(*INK*)
(*************************************************************************************************)
FOR iL_Counter := 1 TO iCIk_NB_INK_PUMPS DO
  (*generate block ads name*)
  aL_Name := sC_Config_I.aC_INKPUMP_NAME;
  IF sC_Config_I.aC_INKPUMP_NAME_DETAIL[iL_Counter] <> '' THEN
    aL_Name := CONCAT(aL_Name, CONCAT(' - ', sC_Config_I.aC_INKPUMP_NAME_DETAIL[iL_Counter]));
  ELSE
    aL_Name := CONCAT(aL_Name, INT_TO_STRING(iL_Counter));
  END_IF
  sAdsIkInkPump[iL_Counter].aO_Name := aL_Name;

  sAdsIkInkPump[iL_Counter].sI_InkPumpSpeedSet.aC_Type := sC_Config_I.aC_INKPUMP_SPEED_TYPE;
  sAdsIkInkPump[iL_Counter].sI_InkPumpSpeedSet.aC_Unit := sC_Config_I.aC_INKPUMP_SPEED_UNIT;
  sAdsIkInkPump[iL_Counter].sI_InkPumpSpeedSet.lC_Min  := sC_Config_I.lL_INKPUMP_SPEED_SET_MIN;
  sAdsIkInkPump[iL_Counter].sI_InkPumpSpeedSet.lC_Max  := sC_Config_I.lL_INKPUMP_SPEED_SET_MAX;
END_FOR

FOR iL_Counter := 1 TO iCIk_NB_HEADERTANK DO
  (*IF bCIk_HEADERTANK_EXIST[iL_Counter] THEN*)
    (*generate block ads name*)
    aL_Name := sC_Config_I.aC_HEADERTANK_NAME;
    IF sC_Config_I.aC_HEADERTANK_NAME_DETAIL[iL_Counter] <> '' THEN
      aL_Name := CONCAT(aL_Name, CONCAT(' - ', sC_Config_I.aC_HEADERTANK_NAME_DETAIL[iL_Counter]));
    ELSE
      aL_Name := CONCAT(aL_Name, INT_TO_STRING(iL_Counter));
    END_IF
    sAdsIkHeaderTank[iL_Counter].aO_Name := aL_Name;

		sAdsIkHeaderTank[iL_Counter].sI_StoragetankAssignment.bC_Exist    := TRUE;
		sAdsIkHeaderTank[iL_Counter].sO_ActStoragetankAssignment.bC_Exist := TRUE;

		(*un-/fill ink*)
		sAdsIkHeaderTank[iL_Counter].bO_EnableFillInkCanEn               := bCIk_HEADERTANK_EXIST[iL_Counter];
		sAdsIkHeaderTank[iL_Counter].bO_EnableUnFillInkCanEn             := bCIk_HEADERTANK_EXIST[iL_Counter];
		sAdsIkHeaderTank[iL_Counter].cO_StatusFillInk.eO_Avbl            := bCIk_HEADERTANK_EXIST[iL_Counter];
		sAdsIkHeaderTank[iL_Counter].cO_StatusUnFillInk.eO_Avbl          := bCIk_HEADERTANK_EXIST[iL_Counter];

		sAdsIkHeaderTank[iL_Counter].sI_ActivateCleaner.bO_CommandCanEx  := bCIk_HEADERTANK_FILL_CLEANER[iL_Counter];
		sAdsIkHeaderTank[iL_Counter].sI_ActivateRefuse.bO_CommandCanEx   := bCIk_HEADERTANK_REFUSE      [iL_Counter];
		sAdsIkHeaderTank[iL_Counter].sI_ActivateExchange.bO_CommandCanEx := FALSE;

		sAdsIkHeaderTank[iL_Counter].sI_ActivateCleaner.bO_CommandExist	 := bCIk_HEADERTANK_FILL_CLEANER[iL_Counter];
		sAdsIkHeaderTank[iL_Counter].sI_ActivateRefuse.bO_CommandExist	 := bCIk_HEADERTANK_REFUSE      [iL_Counter];
		sAdsIkHeaderTank[iL_Counter].sI_ActivateExchange.bO_CommandExist := FALSE;

    sAdsIkHeaderTank[iL_Counter].sI_CommandChange.bO_CommandExist    := bCIk_HEADERTANK_CHANGE      [iL_Counter];

		(*error ack exist*)
		sAdsIkHeaderTank[iL_Counter].sI_AckFillInk.bO_CommandExist       := TRUE;

		(*tank heater*)
		sAdsIkHeaderTank[iL_Counter].sI_TankHeaterSet.bC_Exist   := FALSE;
		sAdsIkHeaderTank[iL_Counter].sI_TankHeaterSet.aC_Type    := sC_Config_I.aC_TEMP_TYPE;
		sAdsIkHeaderTank[iL_Counter].sI_TankHeaterSet.aC_Unit    := sC_Config_I.aC_TEMP_UNIT;
		sAdsIkHeaderTank[iL_Counter].sI_TankHeaterSet.fC_Min     := sC_Config_I.fL_TEMP_SET_VAL_MIN;
		sAdsIkHeaderTank[iL_Counter].sI_TankHeaterSet.fC_Max     := sC_Config_I.fL_TEMP_SET_VAL_MAX;

		sAdsIkHeaderTank[iL_Counter].sO_TankHeaterAct.bC_Exist   := FALSE;
		sAdsIkHeaderTank[iL_Counter].sO_TankHeaterAct.aC_Type    := sC_Config_I.aC_TEMP_TYPE;
		sAdsIkHeaderTank[iL_Counter].sO_TankHeaterAct.aC_Unit    := sC_Config_I.aC_TEMP_UNIT;
    sAdsIkHeaderTank[iL_Counter].sO_TankHeaterAct.fC_Min     := sC_Config_I.fL_TEMP_ACT_VAL_MIN;
    sAdsIkHeaderTank[iL_Counter].sO_TankHeaterAct.fC_Max     := sC_Config_I.fL_TEMP_ACT_VAL_MAX;

		sAdsIkHeaderTank[iL_Counter].bO_EnableTankHeaterCanEn    := FALSE;
		sAdsIkHeaderTank[iL_Counter].cO_StatusTankHeater.eO_Avbl := FALSE;
	(*END_IF*)
END_FOR

FOR iL_Counter := 1 TO iCIk_NB_HEADERTANK_GROUP DO
  (*generate block ads name*)
  aL_Name := sC_Config_I.aC_HEADERTANKGROUP_NAME;
  IF sC_Config_I.aC_HEADERTANKGROUP_NAME_DETAIL[iL_Counter] <> '' THEN
    aL_Name := CONCAT(aL_Name, CONCAT(' - ', sC_Config_I.aC_HEADERTANKGROUP_NAME_DETAIL[iL_Counter]));
  ELSE
    aL_Name := CONCAT(aL_Name, INT_TO_STRING(iL_Counter));
  END_IF
  sAdsIkHeaderTankGroup[iL_Counter].aO_Name := aL_Name;

  sAdsIkHeaderTankGroup[iL_Counter].sI_CommandChangeInk.bO_CommandExist := TRUE;
  sAdsIkHeaderTankGroup[iL_Counter].sI_CommandChangeInk.bO_CommandCanEx := TRUE;
  sAdsIkHeaderTankGroup[iL_Counter].sI_CommandEmptyInk.bO_CommandExist  := FALSE;
  sAdsIkHeaderTankGroup[iL_Counter].sI_CommandEmptyInk.bO_CommandCanEx  := FALSE;
END_FOR


(*TEMP*)
(*************************************************************************************************)
FOR iL_Counter := 1 TO iCIk_NB_TEMP_CONTR DO
  (*generate block ads name*)
  aL_Name := sC_Config_I.aC_TEMP_NAME;
  IF sC_Config_I.aC_TEMP_NAME_DETAIL[iL_Counter] <> '' THEN
    aL_Name := CONCAT(aL_Name, CONCAT(' - ', sC_Config_I.aC_TEMP_NAME_DETAIL[iL_Counter]));
  ELSE
    aL_Name := CONCAT(aL_Name, INT_TO_STRING(iL_Counter));
  END_IF
  sAdsIkHeater[iL_Counter].aO_Name := aL_Name;

  sAdsIkHeater[iL_Counter].sI_HeaterSet.aC_Type    := sC_Config_I.aC_TEMP_TYPE;
  sAdsIkHeater[iL_Counter].sI_HeaterSet.aC_Unit    := sC_Config_I.aC_TEMP_UNIT;
  sAdsIkHeater[iL_Counter].sI_HeaterSet.fC_Min     := sC_Config_I.fL_TEMP_SET_VAL_MIN;
  sAdsIkHeater[iL_Counter].sI_HeaterSet.fC_Max     := sC_Config_I.fL_TEMP_SET_VAL_MAX;

  sAdsIkHeater[iL_Counter].sO_HeaterAct.aC_Type    := sC_Config_I.aC_TEMP_TYPE;
  sAdsIkHeater[iL_Counter].sO_HeaterAct.aC_Unit    := sC_Config_I.aC_TEMP_UNIT;
  sAdsIkHeater[iL_Counter].sO_HeaterAct.fC_Min     := sC_Config_I.fL_TEMP_ACT_VAL_MIN;
  sAdsIkHeater[iL_Counter].sO_HeaterAct.fC_Max     := sC_Config_I.fL_TEMP_ACT_VAL_MAX;

  sAdsIkHeater[iL_Counter].bO_EnableHeaterCanEn    := TRUE;
  sAdsIkHeater[iL_Counter].cO_StatusHeater.eO_Avbl := TRUE;
END_FOR


(* STORAGE TANK *)
(**********************************************************************************)
FOR iL_Counter := 1 TO iCIk_NB_INKSTORAGE_TANK DO
  (*generate block ads name*)
  aL_Name := sC_Config_I.aC_STORAGETANK_NAME;
  IF sC_Config_I.aC_STORAGETANK_NAME_DETAIL[iL_Counter] <> '' THEN
    aL_Name := CONCAT(aL_Name, CONCAT(' - ', sC_Config_I.aC_STORAGETANK_NAME_DETAIL[iL_Counter]));
  ELSE
    aL_Name := CONCAT(aL_Name, INT_TO_STRING(iL_Counter));
  END_IF
  sAdsIkInkStorageTank[iL_Counter].aO_Name := aL_Name;

  (*Special storage tank for conservation*)
  IF sC_Config_I.aC_STORAGETANK_NAME_DETAIL[iL_Counter] = sC_Config_I.aC_STORAGETANK_CONSERVATION THEN
    sAdsIkInkStorageTank[iL_Counter].bO_EnableStorageTankCanEn             := FALSE;
    sAdsIkInkStorageTank[iL_Counter].cO_StatusStorageTank.eO_Avbl          := FALSE;
    sAdsIkInkStorageTank[iL_Counter].sI_EnableMaintenance.bO_CommandCanEx  := FALSE;
    sAdsIkInkStorageTank[iL_Counter].sI_EnableMaintenance.bO_CommandExist  := FALSE;
    sAdsIkInkStorageTank[iL_Counter].fO_StorageTankLevelLiter.bC_Exist     := FALSE;
    sAdsIkInkStorageTank[iL_Counter].sI_MaintenanceTimeout.bC_Exist        := FALSE;
    
    (*Varnish parameter*)
    sAdsIkInkStorageTank[iL_Counter].bO_InkParameterExist                  := FALSE;
    sAdsIkInkStorageTank[iL_Counter].sI_InkParameter.sTemperature.aC_Type  := sC_Config_I.aC_TEMP_TYPE;
    sAdsIkInkStorageTank[iL_Counter].sI_InkParameter.sTemperature.aC_Unit  := sC_Config_I.aC_TEMP_UNIT;
    sAdsIkInkStorageTank[iL_Counter].sI_InkParameter.sTemperature.fC_Min   := sC_Config_I.fL_TEMP_SET_VAL_MIN;
    sAdsIkInkStorageTank[iL_Counter].sI_InkParameter.sTemperature.fC_Max   := sC_Config_I.fL_TEMP_SET_VAL_MAX;
    sAdsIkInkStorageTank[iL_Counter].sI_InkParameter.sMeniscus.aC_Type     := sC_Config_I.aC_SUB_MENC_PRESS_TYPE;
    sAdsIkInkStorageTank[iL_Counter].sI_InkParameter.sMeniscus.aC_Unit     := sC_Config_I.aC_SUB_MENC_PRESS_UNIT;
    sAdsIkInkStorageTank[iL_Counter].sI_InkParameter.sMeniscus.fC_Min      := sC_Config_I.fL_SUB_MENC_PRESS_SET_MIN;
    sAdsIkInkStorageTank[iL_Counter].sI_InkParameter.sMeniscus.fC_Max      := sC_Config_I.fL_SUB_MENC_PRESS_SET_MAX;
    sAdsIkInkStorageTank[iL_Counter].sI_InkParameter.sDensity.aC_Unit      := sC_Config_I.aC_STORAGETANK_DENSITY;
    sAdsIkInkStorageTank[iL_Counter].sI_InkParameter.sViscosity.aC_Unit    := sC_Config_I.aC_STORAGETANK_VISCOSITY;

    sAdsIkInkStorageTank[iL_Counter].sI_EnableBalance.bO_CommandCanEx      := FALSE;
    sAdsIkInkStorageTank[iL_Counter].sI_EnableBalance.bO_CommandExist      := FALSE;
    sAdsIkInkStorageTank[iL_Counter].cO_StatusBalance.eO_Avbl              := FALSE;
    sAdsIkInkStorageTank[iL_Counter].bO_SetZeroCanEx                       := FALSE;
  ELSE
    sAdsIkInkStorageTank[iL_Counter].bI_EnableStorageTank                  := TRUE;
    sAdsIkInkStorageTank[iL_Counter].bO_EnableStorageTankCanEn             := TRUE;
    sAdsIkInkStorageTank[iL_Counter].cO_StatusStorageTank.eO_Avbl          := FALSE;
  
    sAdsIkInkStorageTank[iL_Counter].sI_EnableMaintenance.bO_CommandCanEx  := TRUE;
    sAdsIkInkStorageTank[iL_Counter].sI_EnableMaintenance.bO_CommandExist  := TRUE;
  
    sAdsIkInkStorageTank[iL_Counter].fO_StorageTankLevelLiter.aC_Type      := sC_Config_I.aC_STORAGETANK_TYPE;
    sAdsIkInkStorageTank[iL_Counter].fO_StorageTankLevelLiter.aC_Unit      := sC_Config_I.aC_STORAGETANK_UNITLITER;
    sAdsIkInkStorageTank[iL_Counter].fO_StorageTankLevelPercent.aC_Type    := sC_Config_I.aC_STORAGETANK_TYPE;
    sAdsIkInkStorageTank[iL_Counter].fO_StorageTankLevelPercent.aC_Unit    := sC_Config_I.aC_STORAGETANK_UNITPERCENT;
  
    sAdsIkInkStorageTank[iL_Counter].sI_MaintenanceTimeout.aC_Type         := sC_Config_I.aC_STORAGETANK_MAINTENANCE_TYPE;
    sAdsIkInkStorageTank[iL_Counter].sI_MaintenanceTimeout.aC_Unit         := sC_Config_I.aC_STORAGETANK_MAINTENANCE_UNIT;
    sAdsIkInkStorageTank[iL_Counter].sI_MaintenanceTimeout.lC_Min          := sC_Config_I.lL_STORAGETANK_MAINTENANCE_SET_MIN;
    sAdsIkInkStorageTank[iL_Counter].sI_MaintenanceTimeout.lC_Max          := sC_Config_I.lL_STORAGETANK_MAINTENANCE_SET_MAX;
  
    (*Varnish parameter*)
    sAdsIkInkStorageTank[iL_Counter].bO_InkParameterExist                  := TRUE;
    sAdsIkInkStorageTank[iL_Counter].sI_InkParameter.sTemperature.aC_Type  := sC_Config_I.aC_TEMP_TYPE;
    sAdsIkInkStorageTank[iL_Counter].sI_InkParameter.sTemperature.aC_Unit  := sC_Config_I.aC_TEMP_UNIT;
    sAdsIkInkStorageTank[iL_Counter].sI_InkParameter.sTemperature.fC_Min   := sC_Config_I.fL_TEMP_SET_VAL_MIN;
    sAdsIkInkStorageTank[iL_Counter].sI_InkParameter.sTemperature.fC_Max   := sC_Config_I.fL_TEMP_SET_VAL_MAX;
    sAdsIkInkStorageTank[iL_Counter].sI_InkParameter.sMeniscus.aC_Type     := sC_Config_I.aC_SUB_MENC_PRESS_TYPE;
    sAdsIkInkStorageTank[iL_Counter].sI_InkParameter.sMeniscus.aC_Unit     := sC_Config_I.aC_SUB_MENC_PRESS_UNIT;
    sAdsIkInkStorageTank[iL_Counter].sI_InkParameter.sMeniscus.fC_Min      := sC_Config_I.fL_SUB_MENC_PRESS_SET_MIN;
    sAdsIkInkStorageTank[iL_Counter].sI_InkParameter.sMeniscus.fC_Max      := sC_Config_I.fL_SUB_MENC_PRESS_SET_MAX;
    sAdsIkInkStorageTank[iL_Counter].sI_InkParameter.sDensity.aC_Unit      := sC_Config_I.aC_STORAGETANK_DENSITY;
    sAdsIkInkStorageTank[iL_Counter].sI_InkParameter.sViscosity.aC_Unit    := sC_Config_I.aC_STORAGETANK_VISCOSITY;
  END_IF
END_FOR;

FOR iL_Counter := 1 TO iCIk_NB_INKSTORAGE_TANK DO
  (*Varnish parameter*)
  IF sAdsIkInkStorageTank[iL_Counter].bO_InkParameterExist THEN
    sAdsIkInkStorageTank[iL_Counter].sI_InkParameter.iScannerId          := sR_RemVar_I.lR_VarParamScannerId[iL_Counter];
    sAdsIkInkStorageTank[iL_Counter].sI_InkParameter.iIndex              := sR_RemVar_I.iR_VarParamIndex    [iL_Counter];
    sAdsIkInkStorageTank[iL_Counter].sI_InkParameter.sTemperature.fI_Val := sR_RemVar_I.fR_VarParamTemp     [iL_Counter];
    sAdsIkInkStorageTank[iL_Counter].sI_InkParameter.sMeniscus.fI_Val    := sR_RemVar_I.fR_VarParamMenc     [iL_Counter];
    sAdsIkInkStorageTank[iL_Counter].sI_InkParameter.aWaveform           := sR_RemVar_I.aR_VarParamWaveform [iL_Counter];
    sAdsIkInkStorageTank[iL_Counter].sI_InkParameter.iTimer              := sR_RemVar_I.iR_VarParamTimer    [iL_Counter];
    sAdsIkInkStorageTank[iL_Counter].sI_InkParameter.sDensity.fI_Val     := sR_RemVar_I.fR_VarParamDensity  [iL_Counter];
    sAdsIkInkStorageTank[iL_Counter].sI_InkParameter.sViscosity.fI_Val   := sR_RemVar_I.fR_VarParamViscosity[iL_Counter];
    sAdsIkInkStorageTank[iL_Counter].sI_InkParameter.iColorId            := sR_RemVar_I.iR_VarParamColorId  [iL_Counter];
    FOR iL_Counter2 := 1 TO 10 DO
      sAdsIkInkStorageTank[iL_Counter].sI_InkParameter.bCompatibility[iL_Counter2] := sR_RemVar_I.bR_VarParamCompatibility[iL_Counter, iL_Counter2];
    END_FOR;
  END_IF
END_FOR;


(* BALANCE *)
(*************************************************************************************************)
(* -------------- init of the channels -------------------- *)
FOR iL_Counter := 1 TO iCIk_NB_INKBALANCE DO
  sAdsIkInkStorageTank[iL_Counter].sI_EnableBalance.bI_Command      := TRUE;
	sAdsIkInkStorageTank[iL_Counter].sI_EnableBalance.bO_CommandCanEx := TRUE;
	sAdsIkInkStorageTank[iL_Counter].sI_EnableBalance.bO_CommandExist := TRUE;
	sAdsIkInkStorageTank[iL_Counter].cO_StatusBalance.eO_Avbl         := TRUE;
	sAdsIkInkStorageTank[iL_Counter].bO_SetZeroCanEx                  := TRUE;

	sAdsIkInkStorageTank[iL_Counter].sI_InkDensitySet.aC_Type         := sC_Config_I.aC_BALANCE_INKDENSITY_TYPE;
	sAdsIkInkStorageTank[iL_Counter].sI_InkDensitySet.aC_Unit         := sC_Config_I.aC_BALANCE_INKDENSITY_UNIT;
	sAdsIkInkStorageTank[iL_Counter].sI_InkDensitySet.fC_Min          := sC_Config_I.aC_BALANCE_INKDENSITY_SET_MIN;
	sAdsIkInkStorageTank[iL_Counter].sI_InkDensitySet.fC_Max          := sC_Config_I.aC_BALANCE_INKDENSITY_SET_MAX;

	sAdsIkInkStorageTank[iL_Counter].sI_CorrectionValue.aC_Type       := sC_Config_I.aC_BALANCE_CORRECTION_TYPE;
	sAdsIkInkStorageTank[iL_Counter].sI_CorrectionValue.aC_Unit       := sC_Config_I.aC_BALANCE_CORRECTION_UNIT;
	sAdsIkInkStorageTank[iL_Counter].sI_CorrectionValue.fC_Min        := sC_Config_I.aC_BALANCE_CORRECTION_SET_MIN;
	sAdsIkInkStorageTank[iL_Counter].sI_CorrectionValue.fC_Max        := sC_Config_I.aC_BALANCE_CORRECTION_SET_MAX;

	sAdsIkInkStorageTank[iL_Counter].sI_WarningLevelSet.aC_Type       := sC_Config_I.aC_BALANCE_WARNINGLEVEL_TYPE;
	sAdsIkInkStorageTank[iL_Counter].sI_WarningLevelSet.aC_Unit       := sC_Config_I.aC_BALANCE_WARNINGLEVEL_UNIT;
	sAdsIkInkStorageTank[iL_Counter].sI_WarningLevelSet.fC_Min        := sC_Config_I.aC_BALANCE_WARNINGLEVEL_SET_MIN;
	sAdsIkInkStorageTank[iL_Counter].sI_WarningLevelSet.fC_Max        := sC_Config_I.aC_BALANCE_WARNINGLEVEL_SET_MAX;

	sAdsIkInkStorageTank[iL_Counter].sI_ErrorlevelSet.aC_Type         := sC_Config_I.aC_BALANCE_ERRORLEVEL_TYPE;
	sAdsIkInkStorageTank[iL_Counter].sI_ErrorlevelSet.aC_Unit         := sC_Config_I.aC_BALANCE_ERRORLEVEL_UNIT;
	sAdsIkInkStorageTank[iL_Counter].sI_ErrorlevelSet.fC_Min          := sC_Config_I.aC_BALANCE_ERRORLEVEL_SET_MIN;
	sAdsIkInkStorageTank[iL_Counter].sI_ErrorlevelSet.fC_Max          := sC_Config_I.aC_BALANCE_ERRORLEVEL_SET_MAX;
END_FOR;


(*************************************************************************************************)
(*Function Blocks Init*)
(*************************************************************************************************)


(*neue Lib: new code*)
(*DEGASSING*)
(*************************************************************************************************)
FOR iL_CounterDgas := 1 TO iCIk_NB_DGAS DO
  iSystemCmd.registerForSleepUpdate(iObserver:=fb_DgasMencContr[iL_CounterDgas]);
  
  fb_DgasMencContr[iL_CounterDgas].iRequestMencMinus       := fb_DgasPumpMinus[iL_CounterDgas];
  fb_DgasMencContr[iL_CounterDgas].iRequestMencPlus        := fb_DgasValvePlus[iL_CounterDgas];
  fb_DgasMencContr[iL_CounterDgas].iPurgeController        := fb_PurgeControllerDummy;  (*PurgeBusy not relevant*)
  fb_DgasMencContr[iL_CounterDgas].pConf                   := sC_Config_I.cC_CONF_DGAS_CONTR;
  fb_DgasMencContr[iL_CounterDgas].mInit( pAdsIf         := ADR(sAdsIkDgas [iL_CounterDgas])        (*> ads reference*)
                                        , pMap           := ADR(sL_BLK_DGAS[iL_CounterDgas]));        (*> mapping definition reference*)
  fb_DgasPumpMinus[iL_CounterDgas].Init( sName := 'Dgas pump');

  (*MainValve K111*)
  iSystemCmd.registerForSleepUpdate(iObserver:=fb_DgasMainValve[iL_CounterDgas]);
  fb_DgasMainValve[iL_CounterDgas].mEnable();
END_FOR;

(*MENISCUS*)
(*************************************************************************************************)
FOR iL_CounterMenc := 1 TO iCIk_NB_MENC DO
  iSystemCmd.registerForSleepUpdate(iObserver:=fb_MeniscusMencContr[iL_CounterMenc]);
  
  fb_MeniscusMencContr[iL_CounterMenc].iRequestMencMinus       := fb_MeniscusValveMinus[iL_CounterMenc];
  fb_MeniscusMencContr[iL_CounterMenc].iRequestMencPlus        := fb_MeniscusValvePlus [iL_CounterMenc];
  fb_MeniscusMencContr[iL_CounterMenc].iPurgeController        := fb_PurgeControllerDummy;  (*PurgeBusy not relevant*)
  fb_MeniscusMencContr[iL_CounterMenc].pConf                   := sC_Config_I.cC_CONF_MENC_CONTR;
  fb_MeniscusMencContr[iL_CounterMenc].mInit( pAdsIf         := ADR(sAdsIkMenc [iL_CounterMenc])        (*> ads reference*)
                                            , pMap           := ADR(sL_BLK_MENC[iL_CounterMenc]));      (*> mapping definition reference*)
END_FOR;
fb_MeniscusPump.Init(sName := 'Main meniscus pump');

(*SUB MENISCUS*)
(*************************************************************************************************)
FOR iL_CounterSubMenc := 1 TO iCIk_NB_SUB_MENC DO
  iSystemCmd.registerForSleepUpdate(iObserver:=fb_MeniscusMencContr[iCIk_NB_MENC + iL_CounterSubMenc]);
  
  fb_MeniscusMencContr[iCIk_NB_MENC + iL_CounterSubMenc].iRequestMencMinus       := fb_MeniscusValveMinus[iCIk_NB_MENC + iL_CounterSubMenc];
  fb_MeniscusMencContr[iCIk_NB_MENC + iL_CounterSubMenc].iRequestMencPlus        := fb_MeniscusValvePlus [iCIk_NB_MENC + iL_CounterSubMenc];
  fb_MeniscusMencContr[iCIk_NB_MENC + iL_CounterSubMenc].iPurgeController        := fb_PurgeControllerDummy;  (*PurgeBusy not relevant*)
  fb_MeniscusMencContr[iCIk_NB_MENC + iL_CounterSubMenc].pConf                   := sC_Config_I.cC_CONF_SUB_MENC_CONTR;
  fb_MeniscusMencContr[iCIk_NB_MENC + iL_CounterSubMenc].mInit( pAdsIf         := ADR(sAdsIkMenc [iCIk_NB_MENC + iL_CounterSubMenc])  (*> ads reference*)
                                                              , pMap           := ADR(sL_BLK_MENC[iCIk_NB_MENC + iL_CounterSubMenc]));  (*> mapping definition reference*)
END_FOR;


(*TEMP*)
(*************************************************************************************************)
(*Headertank heater*)
FOR iL_Counter := 1 TO iCIk_NB_TEMP_HYS DO
  iSystemCmd.registerForSleepUpdate(iObserver:=fb_TempControllerHys[iL_Counter]);
  iSystemCmd.registerForEmergencyUpdate(iObserver:=fb_TempControllerHys[iL_Counter]);

  fb_TempControllerHys[iL_Counter].mInit( pAdsIf         := ADR(sAdsIkHeater[iL_Counter]));           (*> ads reference*)
  fb_TempControllerHys[iL_Counter].mEnable();
END_FOR;


(*PURGE*)
(*************************************************************************************************)
FOR iL_Counter := 1 TO iCIk_NB_PURGE_CONTR DO
  fb_PurgeController[iL_Counter].iMachineInk       := PRG_MACHINE.iMachineInk[iL_Counter];
  fb_PurgeController[iL_Counter].iSubMencNeg       := fb_MeniscusMencContr[bCIk_MAP_PURGE_CONTR_SEQ_MENC_NEG[iL_Counter]];
  fb_PurgeController[iL_Counter].iSubMencPos       := fb_MeniscusMencContr[bCIk_MAP_PURGE_CONTR_SEQ_MENC_POS[iL_Counter]];
  fb_PurgeController[iL_Counter].pActivateSequence := bCIk_PURGE_CONTR_SEQUENCE[iL_Counter];
  fb_PurgeController[iL_Counter].pAirOk            := TRUE;
  fb_PurgeController[iL_Counter].mInit( pAdsIf         := ADR(sAdsIkPurgeController[iL_Counter])  (*> ads reference*)
                                      , pMap           := ADR(sL_BLK_PURGE_CONTR   [iL_Counter]));  (*> mapping definition reference*)
END_FOR

FOR iL_Counter := 1 TO iCIk_NB_PURGE_GROUP DO
  fb_PurgeGroup     [iL_Counter].mInit( pAdsIf         := ADR(sAdsIkPurgeGroup  [iL_Counter])     (*> ads reference*)
                                      , pMap           := ADR(sL_BLK_PURGE_GROUP[iL_Counter]));     (*> mapping definition reference*)

  IF cL_State = cL_INIT_PRG THEN
    fb_PurgeController[cCIk_MAP_PURGE_GROUP_CONTR[iL_Counter]].mRegisterGroup(fb_PurgeGroup[iL_Counter]);
  END_IF
END_FOR


(*VACUUM PUMP*)
(*************************************************************************************************)


(*INK*)
(*************************************************************************************************)
FOR iL_Counter := 1 TO iCIk_NB_HEADERTANK DO
  fb_FillInkVarnish[iL_Counter].cI_Conf           := sC_Config_I.cC_CONF_INK_SUPPLY_UNIT;

  fb_Headertank[iL_Counter].bI_HeadertankExist    := bCIk_HEADERTANK_EXIST[iL_Counter];

  (*Messaging*)
  (*Config FB_HEADERTANK_UNIT*)
  fb_Headertank[iL_Counter].pC_MsgInterface       := ADR(sAdsIkHeaderTank[iL_Counter].sO_Message);
  fb_Headertank[iL_Counter].iC_BlockId            := eIk_BLK_HEADERTANK;
  fb_Headertank[iL_Counter].Init();

  (*Config FB_INK_SUPPLY_UNIT*)
  (*Only dummy, messaging is now handled by fb_Headertank*)
  fb_FillInkVarnish[iL_Counter].pC_MsgInterface   := ADR(sAdsIkDummy[1].sO_Message);  (*Only dummy, messages are not used in this FB*)
  fb_FillInkVarnish[iL_Counter].iC_BlockId        := 0;                               (*Messages are not used in this FB*)
  fb_FillInkVarnish[iL_Counter].Init();

  (*Circulation ink controller*)
  iSystemCmd.registerForSleepUpdate(iObserver:=fb_CirculationInk[iL_Counter]);
  
  fb_CirculationInk[iL_Counter].iPurgeController := fb_PurgeController[iCIk_MAP_HEADERTANK_PURGE_CONTR[iL_Counter]];
  fb_CirculationInk[iL_Counter].iMencController  := fb_MeniscusMencContr[iCIk_MAP_HEADERTANK_MENC_STA[iL_Counter]];
  fb_CirculationInk[iL_Counter].pName            := sC_Config_I.aC_HEADERTANK_NAME_DETAIL[iL_Counter];
END_FOR


(* STORAGE TANK *)
(**********************************************************************************)
FOR iL_Counter := 1 TO iCIk_NB_INKSTORAGE_TANK DO
  (*Messaging*)
  (*Config FB_STORAGETANK_UNIT*)
  fb_Storagetank[iL_Counter].pC_MsgInterface       := ADR(sAdsIkDummy[1].sO_Message);  (*ADR(sAdsIkInkStorageTank[iL_Counter].sO_Message);*)
  fb_Storagetank[iL_Counter].iC_BlockId            := eIk_BLK_INKSTORAGE_TANK;
  fb_Storagetank[iL_Counter].Init();

  (*Messaging*)
  sL_MsgConfigStorage[iL_Counter].bI_Enable       := TRUE;
  sL_MsgConfigStorage[iL_Counter].pI_FbMsgHandler := ADR(fB_BalanceMsgHandler[iL_Counter]);

  fB_BalanceMsgHandler[iL_Counter].pI_MsgQueue    := ADR(fB_MsgQueueStorage[iL_Counter]);

  fB_MsgQueueStorage[iL_Counter].pI_MsgInterface  := ADR(sAdsIkInkStorageTank[iL_Counter].sO_Message);
  fB_MsgQueueStorage[iL_Counter].cI_MaxElement    := 5;

  FOR iL_Counter2 := 1 TO iCIk_NB_BALANCE_MSG DO
    fB_BalanceMsg[iL_Counter, iL_Counter2].pI_MsgConfig   := ADR(sL_MsgConfigStorage[iL_Counter]);
    fB_BalanceMsg[iL_Counter, iL_Counter2].iI_MsgLocation := iL_Counter;
  END_FOR;

  fB_BalanceMsg[iL_Counter,  1].iI_MsgNumber      := eCIk_STOR_BAL_SEND;
  fB_BalanceMsg[iL_Counter,  2].iI_MsgNumber      := eCIk_STOR_BAL_RECEIVE;
  fB_BalanceMsg[iL_Counter,  3].iI_MsgNumber      := eCIk_STOR_BAL_MOTION;
  fB_BalanceMsg[iL_Counter,  4].iI_MsgNumber      := eCIk_STOR_BAL_NOCONNECT;
  fb_BalanceMsg[iL_Counter,  5].iI_MsgNumber      := eCIk_STOR_BAL_BUFFERFULL;
  fb_BalanceMsg[iL_Counter,  6].iI_MsgNumber      := eCIk_STOR_BAL_FRAMEFAULT;
  fb_BalanceMsg[iL_Counter,  7].iI_MsgNumber      := eCIk_STOR_BAL_OVERRUN;
  fb_BalanceMsg[iL_Counter,  8].iI_MsgNumber      := eCIk_STOR_LVL_WARNING;
  fb_BalanceMsg[iL_Counter,  9].iI_MsgNumber      := eCIk_STOR_LVL_ERROR;
  fb_BalanceMsg[iL_Counter, 10].iI_MsgNumber      := eCIk_STOR_TANK_MISSING;
  fb_BalanceMsg[iL_Counter, 11].iI_MsgNumber      := eCIk_STOR_TANK_MIXER_NOT_WORKING;
  fb_BalanceMsg[iL_Counter, 12].iI_MsgNumber      := eCIk_STOR_LVL_INFO;
  fb_BalanceMsg[iL_Counter, 13].iI_MsgNumber      := eCIk_STOR_SCAN_NEED;
  fb_BalanceMsg[iL_Counter, 14].iI_MsgNumber      := eCIk_STOR_SCAN_FALSE;
  fb_BalanceMsg[iL_Counter, 15].iI_MsgNumber      := eCIk_STOR_HT_ASSIGNMENT;
END_FOR;


(* BALANCE *)
(*************************************************************************************************)
(* -------------- init of the channels -------------------- *)
FOR iL_Counter := 1 TO iCIk_NB_INKBALANCE DO
  fb_Balance[iL_Counter].pI_BalanceOffset := ADR(fL_BalanceOffset[iL_Counter]);

  fb_BalanceLink.pI_ZeroPointerErr                 := ADR(nConvError);
  fb_BalanceLink.iI_UsedBalanceMux                 := iCIk_NB_BALANCE_MUX;
  fb_BalanceLink.bI_ZS_SelectedChannel[iL_Counter] := FALSE;
  fb_BalanceLink.bI_CS_SelectedChannel[iL_Counter] := FALSE;

  fb_BalanceLink( cI_MapBalanceBalanceMux     := cCIk_MAP_BALANCE_BALANCE_MUX
                , cI_MapBalanceBalanceChannel := cCIk_MAP_BALANCE_BALANCE_CHANNEL);
  
END_FOR;


  
(*************************************************************************************************)
(*ADS blocks mapping*)
(*************************************************************************************************)

(*Recipe read/write*)
(*************************************************************************************************)
IF cL_State = cL_INIT_PRG THEN
  pFbRecipeMngr := PRG_SYSTEMBASE.registerRecipe(
    aI_RecipePath           := CONCAT(aC_PlcConfigPath, aC_PlcRecipeSubPath),
    aI_RecipeDefinitionName := sC_Ads_Info.aType  (*is set in Mapping*)
  );
 
  (* -- BlockId saving ----------------------------------------------------------------------------*)
  PRG_SYSTEMBASE.fbBlockIdSave.registerModule(
    aI_StoragePath := CONCAT(aC_PlcConfigPath, aC_PlcBlockIdSubPath),
    pI_Ads_Info    := ADR(sC_Ads_Info)
  );
END_IF


(********************************* END OF ACTION *************************************************)
END_ACTION

ACTION Mapping:
(*************************************************************************************************)
(*ADS blocks mapping definition*)
(*************************************************************************************************)
(*mapping of each block with his parents, unique type and index*)

(*purge controller*)
FOR iL_Counter := 1 TO iCIk_NB_PURGE_CONTR DO
  IF bCIk_PURGE_CONTR_EXIST[iL_Counter] THEN
    (*purge controller -> root*)
		sL_BLK_PURGE_CONTR[iL_Counter].iPMaps[1]    := FC_ADD_MAP(eSys_BLK_ROOT, 1);
  END_IF;
END_FOR;

(*purge group*)
FOR iL_Counter := 1 TO iCIk_NB_PURGE_GROUP DO
  IF bCIk_PURGE_GROUP_EXIST[iL_Counter] THEN
    (*purge group -> purge controller*)
    sL_BLK_PURGE_GROUP[iL_Counter].iPMaps[1]      := FC_ADD_MAP(eIk_BLK_PURGE_CONTROLLER, cCIk_MAP_PURGE_GROUP_CONTR[iL_Counter]);
  END_IF;
END_FOR;

(*dgas*)
FOR iL_Counter := 1 TO iCIk_NB_DGAS DO
  (*dgas -> root*)
  sL_BLK_DGAS[iL_Counter].iPMaps[1]             := FC_ADD_MAP(eSys_BLK_ROOT, 1);
  (*dgas -> purge*)
(*sL_BLK_DGAS[iL_Counter].iPMaps[2]             := FC_ADD_MAP(eIk_BLK_PURGE_CONTROLLER, 1);
  sL_BLK_DGAS[iL_Counter].iPMaps[3]             := FC_ADD_MAP(eIk_BLK_PURGE_CONTROLLER, 2);*)
END_FOR;

(*menc*)
FOR iL_Counter := 1 TO iCIk_NB_MENC DO
  (*main menc -> root*)
  sL_BLK_MENC[iL_Counter].iPMaps[1]             := FC_ADD_MAP(eSys_BLK_ROOT, 1);
END_FOR;
FOR iL_Counter := 1 TO iCIk_NB_SUB_MENC DO
  (*sub menc -> menc*)
  sL_BLK_MENC[iCIk_NB_MENC + iL_Counter].iPMaps[1] := FC_ADD_MAP(eIk_BLK_MENC, iCIk_MAP_SUB_MENC_MAIN_MENC[iL_Counter]);
  (*sub menc -> header tank group*)
  sL_BLK_MENC[iCIk_NB_MENC + iL_Counter].iPMaps[2] := FC_ADD_MAP(eIk_BLK_HEADERTANK_GROUP, iCIk_MAP_SUB_MENC_HTG[iL_Counter]);
END_FOR;

(*ink storage tank*)
FOR iL_Counter := 1 TO iCIk_NB_INKSTORAGE_TANK DO
  IF bCIk_INKSTORAGE_TANK_EXIST[iL_Counter] THEN
    (*ink storage tank -> root*)
    sL_BLK_INKSTORAGE_TANK[iL_Counter].iPMaps[1] := FC_ADD_MAP(eSys_BLK_ROOT, 1);
  END_IF;
END_FOR;

(*header tank group*)
FOR iL_Counter := 1 TO iCIk_NB_HEADERTANK_GROUP DO
  (*header tank group -> storage tank*)
  sL_BLK_HEADERTANK_GROUP[iL_Counter].iPMaps[1]   := FC_ADD_MAP(eIk_BLK_INKSTORAGE_TANK, 1);
  sL_BLK_HEADERTANK_GROUP[iL_Counter].iPMaps[2]   := FC_ADD_MAP(eIk_BLK_INKSTORAGE_TANK, 2);
END_FOR;

(*header tank*)
FOR iL_Counter := 1 TO iCIk_NB_HEADERTANK DO
  IF bCIk_HEADERTANK_EXIST[iL_Counter] THEN
    (*header tank -> storage tank*)
    sL_BLK_HEADERTANK[iL_Counter].iPMaps[1]       := FC_ADD_MAP(eIk_BLK_INKSTORAGE_TANK, 1);
    sL_BLK_HEADERTANK[iL_Counter].iPMaps[2]       := FC_ADD_MAP(eIk_BLK_INKSTORAGE_TANK, 2);

    (*header tank -> meniscus*)
    sL_BLK_HEADERTANK[iL_Counter].iPMaps[3]       := FC_ADD_MAP(eIk_BLK_MENC, iCIk_MAP_HEADERTANK_MENC_STA[iL_Counter]);

    (*header tank -> header tank group*)
    sL_BLK_HEADERTANK[iL_Counter].iPMaps[4]       := FC_ADD_MAP(eIk_BLK_HEADERTANK_GROUP, iCIk_MAP_HEADERTANK_HT_GROUP[iL_Counter]);
  END_IF;
END_FOR;

(*heater*)
FOR iL_Counter := 1 TO iCIk_NB_TEMP_CONTR DO
  (*heater -> root*)
  sL_BLK_HEATER[iL_Counter].iPMaps[1]           := FC_ADD_MAP(eSys_BLK_ROOT, 1);
  (*heater -> group*)
  sL_BLK_HEATER[iL_Counter].iPMaps[2]           := FC_ADD_MAP(ePr_BLK_PG, iCIk_MAP_TEMP_PG[iL_Counter]);
END_FOR;


(*ADS blocks configuration & information*)
(*************************************************************************************************)
sC_Ads_Info.bReady   := FALSE;
sC_Ads_Info.aType    := 'PRG_INK';
sC_Ads_Info.iVersion := 010000;        (*1.0.0*)
sC_Ads_Info.iType    := eMOD_INK;

sMappingInfo.init(lModId:=TO_UINT(eMOD_INK)); 
sMappingInfo.addBlkAry( iAdsBlockType := TO_UINT(eIk_BLK_PURGE_CONTROLLER), aAdsBlockName := 'sAdsIkPurgeController', iAdsBlockVersion:= INT_TO_UINT(sAdsIkPurgeController[1].iO_Version), iNbrBlocks := SIZEOF(sL_BLK_PURGE_CONTR)     / SIZEOF(sL_BLK_PURGE_CONTR[1]),     pBlockArray := ADR(sL_BLK_PURGE_CONTR));
sMappingInfo.addBlkAry( iAdsBlockType := TO_UINT(eIk_BLK_PURGE_GROUP),      aAdsBlockName := 'sAdsIkPurgeGroup',      iAdsBlockVersion:= INT_TO_UINT(sAdsIkPurgeGroup[1].iO_Version),      iNbrBlocks := SIZEOF(sL_BLK_PURGE_GROUP)     / SIZEOF(sL_BLK_PURGE_GROUP[1]),     pBlockArray := ADR(sL_BLK_PURGE_GROUP));
sMappingInfo.addBlkAry( iAdsBlockType := TO_UINT(eIk_BLK_DGAS),             aAdsBlockName := 'sAdsIkDgas',            iAdsBlockVersion:= INT_TO_UINT(sAdsIkDgas[1].iO_Version),            iNbrBlocks := SIZEOF(sL_BLK_DGAS)            / SIZEOF(sL_BLK_DGAS[1]),            pBlockArray := ADR(sL_BLK_DGAS));
sMappingInfo.addBlkAry( iAdsBlockType := TO_UINT(eIk_BLK_MENC),             aAdsBlockName := 'sAdsIkMenc',            iAdsBlockVersion:= INT_TO_UINT(sAdsIkMenc[1].iO_Version),            iNbrBlocks := SIZEOF(sL_BLK_MENC)            / SIZEOF(sL_BLK_MENC[1]),            pBlockArray := ADR(sL_BLK_MENC));
sMappingInfo.addBlkAry( iAdsBlockType := TO_UINT(eIk_BLK_HEADERTANK_GROUP), aAdsBlockName := 'sAdsIkHeaderTankGroup', iAdsBlockVersion:= INT_TO_UINT(sAdsIkHeaderTankGroup[1].iO_Version), iNbrBlocks := SIZEOF(sL_BLK_HEADERTANK_GROUP)/ SIZEOF(sL_BLK_HEADERTANK_GROUP[1]),pBlockArray := ADR(sL_BLK_HEADERTANK_GROUP));
sMappingInfo.addBlkAry( iAdsBlockType := TO_UINT(eIk_BLK_HEADERTANK),       aAdsBlockName := 'sAdsIkHeaderTank',      iAdsBlockVersion:= INT_TO_UINT(sAdsIkHeaderTank[1].iO_Version),      iNbrBlocks := SIZEOF(sL_BLK_HEADERTANK)      / SIZEOF(sL_BLK_HEADERTANK[1]),      pBlockArray := ADR(sL_BLK_HEADERTANK));
sMappingInfo.addBlkAry( iAdsBlockType := TO_UINT(eIk_BLK_INKSTORAGE_TANK),  aAdsBlockName := 'sAdsIkInkStorageTank',  iAdsBlockVersion:= INT_TO_UINT(sAdsIkInkStorageTank[1].iO_Version),  iNbrBlocks := SIZEOF(sL_BLK_INKSTORAGE_TANK) / SIZEOF(sL_BLK_INKSTORAGE_TANK[1]), pBlockArray := ADR(sL_BLK_INKSTORAGE_TANK));
sMappingInfo.addBlkAry( iAdsBlockType := TO_UINT(eIk_BLK_INKPUMP),          aAdsBlockName := 'sAdsIkInkPump',         iAdsBlockVersion:= INT_TO_UINT(sAdsIkInkPump[1].iO_Version),         iNbrBlocks := SIZEOF(sL_BLK_INKPUMP)         / SIZEOF(sL_BLK_INKPUMP[1]),         pBlockArray := ADR(sL_BLK_INKPUMP));
sMappingInfo.addBlkAry( iAdsBlockType := TO_UINT(eIk_BLK_HEATER),           aAdsBlockName := 'sAdsIkHeater',          iAdsBlockVersion:= INT_TO_UINT(sAdsIkHeater[1].iO_Version),          iNbrBlocks := SIZEOF(sL_BLK_HEATER)          / SIZEOF(sL_BLK_HEATER[1]),          pBlockArray := ADR(sL_BLK_HEATER));
sMappingInfo.bReady := TRUE;

(********************************* END OF ACTION *************************************************)
END_ACTION

ACTION RemVar:
(*************************************************************************************************)
(********************************* READING REMANENT VARIABLES ************************************)
(*************************************************************************************************)
IF bL_RemVar_Init THEN

  (*load initial values if pattern was invalid*)
  IF sR_RemVar_I.aL_Pattern <> 16#ABCD THEN

    (*initial very boot values of project*)
    sR_RemVar_I.aL_Pattern := 16#ABCD;

    (*TODO add boot/config values*)

    (*DEGASSING*)
    (*************************************************************************************************)
    FOR iL_Counter := 1 TO iCIk_NB_DGAS DO
      sAdsIkDgas[iL_Counter].sI_PressSet.fI_Val             := -400;   (*mbar*)
    END_FOR;


    (*MENISCUS*)
    (*************************************************************************************************)
    (*Main*)
    sAdsIkMenc[1].sI_PressSet.fI_Val                        := sC_Config_I.fL_MENC1_PRESS_INITVAL;       (*mbar*)
    (*Sub*)
    sAdsIkMenc[2].sI_PressSet.fI_Val                        := sC_Config_I.fL_SUB_MENC1_PRESS_INITVAL;   (*mbar*)
    sAdsIkMenc[3].sI_PressSet.fI_Val                        := sC_Config_I.fL_SUB_MENC2_PRESS_INITVAL;   (*mbar*)

    (*Init rem var*)
    FOR iL_CounterMenc := 1 TO iCIk_NB_MENC DO
      fb_MeniscusMencContr[iL_CounterMenc].mInitRemVar( IfConvAdsTtLocal := sC_Config_I.fL_MENC_CONV_ADS_TO_LCL
                                                      , IfPressSetMin    := sC_Config_I.fL_MENC_PRESS_SET_MIN
                                                      , IfPressSetMax    := sC_Config_I.fL_MENC_PRESS_SET_MAX
                                                      , IfPressActMin    := sC_Config_I.fL_MENC_PRESS_ACT_MIN
                                                      , IfPressActMax    := sC_Config_I.fL_MENC_PRESS_ACT_MAX
                                                      , IfTolSmall       := sC_Config_I.fL_MENC_TOL_SMALL
                                                      , IfTolBig         := sC_Config_I.fL_MENC_TOL_BIG);
    END_FOR;
    FOR iL_CounterSubMenc := 1 TO iCIk_NB_SUB_MENC DO
      (*Special for sub men white pos*)
      IF sC_Config_I.aC_SUB_MENC_NAME_DETAIL[iL_CounterSubMenc] = 'Sub White pos' THEN
        fb_MeniscusMencContr[iCIk_NB_MENC + iL_CounterSubMenc].mInitRemVar( IfConvAdsTtLocal := sC_Config_I.fL_SUB_MENC_CONV_ADS_TO_LCL
                                                                          , IfPressSetMin    :=  -2.0
                                                                          , IfPressSetMax    := 120.0
                                                                          , IfPressActMin    :=  -2.0
                                                                          , IfPressActMax    := 120.0
                                                                          , IfTolSmall       := sC_Config_I.fL_SUB_MENC_TOL_SMALL
                                                                          , IfTolBig         := sC_Config_I.fL_SUB_MENC_TOL_BIG);
      ELSE
        fb_MeniscusMencContr[iCIk_NB_MENC + iL_CounterSubMenc].mInitRemVar( IfConvAdsTtLocal := sC_Config_I.fL_SUB_MENC_CONV_ADS_TO_LCL
                                                                          , IfPressSetMin    := sC_Config_I.fL_SUB_MENC_PRESS_SET_MIN
                                                                          , IfPressSetMax    := sC_Config_I.fL_SUB_MENC_PRESS_SET_MAX
                                                                          , IfPressActMin    := sC_Config_I.fL_SUB_MENC_PRESS_ACT_MIN
                                                                          , IfPressActMax    := sC_Config_I.fL_SUB_MENC_PRESS_ACT_MAX
                                                                          , IfTolSmall       := sC_Config_I.fL_SUB_MENC_TOL_SMALL
                                                                          , IfTolBig         := sC_Config_I.fL_SUB_MENC_TOL_BIG);
			END_IF
    END_FOR;
    
    (*INK*)
    (*************************************************************************************************)
    (*varnish*)
    FOR iL_Counter:= 1 TO iCIk_NB_HEADERTANK DO
      sAdsIkHeaderTank[iL_Counter].bI_FillModeAuto          := TRUE;
      sAdsIkHeaderTank[iL_Counter].bI_EnableRamp            := FALSE;
    END_FOR

    
    (*MAINTENANCE*)
    (*************************************************************************************************)
    (*VISU SETTINGS*)
		wIDp_MinSpeedFillInkPumpVarnish                         := 10;     (*%*)
		wIDp_MaxSpeedFillInkPumpVarnish                         := 100;    (*%*)
		wIDP_AnalogMinDigitVarnish                              := 0;
		wIDP_AnalogMaxDigitVarnish                              := 16383;

    lL_TimeReturnFlow                                       := 90;     (*s*)
    lL_TimeBlowOut                                          := 130;    (*s*)
    lL_TimeEmptyCleaner                                     := 60;     (*s*)
    lL_TimeWarnExchange                                     := 6;      (*h*)

    
    (*TEMP*)
    (*************************************************************************************************)
    FOR iL_Counter := 1 TO iCIk_NB_TEMP_CONTR DO
      sAdsIkHeater[iL_Counter].sI_HeaterSet.fI_Val          := 50;    (*°C*)
    END_FOR

    
    (*PURGE*)
    (*************************************************************************************************)
    sAdsIkPurgeController[1].bI_Enable                      := TRUE;

    
